LIN {X 0,Y 523.877,Z 238.227,A -85,B 0,C 180,E1 -4906.892,E2 -4906.892} C_VEL
LIN {X 0,Y 523.199,Z 238.314,A -85,B 0,C 180,E1 -4907.534,E2 -4907.534} C_VEL
LIN {X 0,Y 520.354,Z 238.667,A -85,B 0,C 180,E1 -4908.575,E2 -4908.575} C_VEL
LIN {X 0,Y 517.963,Z 238.966,A -85,B 0,C 180,E1 -4909.414,E2 -4909.414} C_VEL
LIN {X 0,Y 516.943,Z 239.092,A -85,B 0,C 180,E1 -4910.062,E2 -4910.062} C_VEL
LIN {X 0,Y 516.862,Z 239.1,A -85,B 0,C 180,E1 -4910.281,E2 -4910.281} C_VEL
LIN {X 0,Y 516.85,Z 239.107,A -85,B 0,C 180,E1 -4913.252,E2 -4913.252} C_VEL
LIN {X 0,Y 516.776,Z 239.117,A -85,B 0,C 180,E1 -4914.685,E2 -4914.685} C_VEL
LIN {X 0,Y 516.776,Z 242.58,A -85,B 0,C 180,E1 -4917.044,E2 -4917.044} C_VEL
LIN {X 0,Y 516.677,Z 246.727,A -85,B 0,C 180,E1 -4919.782,E2 -4919.782} C_VEL
LIN {X 0,Y 516.622,Z 250.843,A -85,B 0,C 180,E1 -4922.45,E2 -4922.45} C_VEL
LIN {X 0,Y 516.599,Z 255.972,A -85,B 0,C 180,E1 -4925.713,E2 -4925.713} C_VEL
LIN {X 0,Y 516.465,Z 260.373,A -85,B 0,C 180,E1 -4928.444,E2 -4928.444} C_VEL
LIN {X 0,Y 516.401,Z 264.484,A -85,B 0,C 180,E1 -4930.936,E2 -4930.936} C_VEL
LIN {X 0,Y 516.361,Z 268.626,A -85,B 0,C 180,E1 -4933.392,E2 -4933.392} C_VEL
LIN {X 0,Y 516.371,Z 273.427,A -85,B 0,C 180,E1 -4936.171,E2 -4936.171} C_VEL
LIN {X 0,Y 518.506,Z 285.677,A -85,B 0,C 180,E1 -4936.553,E2 -4936.553} C_VEL
LIN {X 0,Y 518.232,Z 298.164,A -85,B 0,C 180,E1 -4937.02,E2 -4937.02} C_VEL
LIN {X 0,Y 518.004,Z 310.503,A -85,B 0,C 180,E1 -4937.651,E2 -4937.651} C_VEL
LIN {X 0,Y 517.663,Z 322.372,A -85,B 0,C 180,E1 -4938.448,E2 -4938.448} C_VEL
LIN {X 0,Y 517.327,Z 332.848,A -85,B 0,C 180,E1 -4939.333,E2 -4939.333} C_VEL
LIN {X 0,Y 517.081,Z 341.406,A -85,B 0,C 180,E1 -4940.218,E2 -4940.218} C_VEL
LIN {X 0,Y 516.859,Z 349.287,A -85,B 0,C 180,E1 -4941.201,E2 -4941.201} C_VEL
LIN {X 0,Y 516.622,Z 356.995,A -85,B 0,C 180,E1 -4942.378,E2 -4942.378} C_VEL
LIN {X 0,Y 516.497,Z 364.061,A -85,B 0,C 180,E1 -4943.751,E2 -4943.751} C_VEL
LIN {X 0,Y 516.313,Z 368.775,A -85,B 0,C 180,E1 -4944.924,E2 -4944.924} C_VEL
LIN {X 0,Y 516.373,Z 372.379,A -85,B 0,C 180,E1 -4946.098,E2 -4946.098} C_VEL
LIN {X 0,Y 516.282,Z 374.246,A -85,B 0,C 180,E1 -4946.879,E2 -4946.879} C_VEL
LIN {X 0,Y 516.261,Z 375.654,A -85,B 0,C 180,E1 -4947.659,E2 -4947.659} C_VEL
LIN {X 0,Y 516.16,Z 377.273,A -85,B 0,C 180,E1 -4949.22,E2 -4949.22} C_VEL
LIN {X 0,Y 516.155,Z 377.51,A -85,B 0,C 180,E1 -4950,E2 -4950} C_VEL
LIN {X 0,Y 516.16,Z 377.327,A -85,B 0,C 180,E1 -4950.78,E2 -4950.78} C_VEL
LIN {X 0,Y 516.261,Z 375.779,A -85,B 0,C 180,E1 -4952.341,E2 -4952.341} C_VEL
LIN {X 0,Y 516.283,Z 374.426,A -85,B 0,C 180,E1 -4953.121,E2 -4953.121} C_VEL
LIN {X 0,Y 516.364,Z 371.563,A -85,B 0,C 180,E1 -4954.293,E2 -4954.293} C_VEL
LIN {X 0,Y 516.404,Z 367.684,A -85,B 0,C 180,E1 -4955.467,E2 -4955.467} C_VEL
LIN {X 0,Y 516.512,Z 362.677,A -85,B 0,C 180,E1 -4956.641,E2 -4956.641} C_VEL
LIN {X 0,Y 516.647,Z 356.375,A -85,B 0,C 180,E1 -4957.818,E2 -4957.818} C_VEL
LIN {X 0,Y 516.859,Z 348.484,A -85,B 0,C 180,E1 -4958.996,E2 -4958.996} C_VEL
LIN {X 0,Y 517.129,Z 338.665,A -85,B 0,C 180,E1 -4960.176,E2 -4960.176} C_VEL
LIN {X 0,Y 517.456,Z 328.368,A -85,B 0,C 180,E1 -4961.16,E2 -4961.16} C_VEL
LIN {X 0,Y 517.77,Z 317.683,A -85,B 0,C 180,E1 -4961.98,E2 -4961.98} C_VEL
LIN {X 0,Y 518.059,Z 307.006,A -85,B 0,C 180,E1 -4962.636,E2 -4962.636} C_VEL
LIN {X 0,Y 518.328,Z 294.474,A -85,B 0,C 180,E1 -4963.227,E2 -4963.227} C_VEL
LIN {X 0,Y 518.333,Z 284.206,A -85,B 0,C 180,E1 -4963.589,E2 -4963.589} C_VEL
LIN {X 0,Y 516.384,Z 273.353,A -85,B 0,C 180,E1 -4963.93,E2 -4963.93} C_VEL
LIN {X 0,Y 516.354,Z 268.778,A -85,B 0,C 180,E1 -4966.608,E2 -4966.608} C_VEL
LIN {X 0,Y 516.396,Z 264.635,A -85,B 0,C 180,E1 -4969.065,E2 -4969.065} C_VEL
LIN {X 0,Y 516.468,Z 260.521,A -85,B 0,C 180,E1 -4971.556,E2 -4971.556} C_VEL
LIN {X 0,Y 516.568,Z 256.141,A -85,B 0,C 180,E1 -4974.279,E2 -4974.279} C_VEL
LIN {X 0,Y 516.591,Z 252.355,A -85,B 0,C 180,E1 -4976.677,E2 -4976.677} C_VEL
LIN {X 0,Y 516.667,Z 248.011,A -85,B 0,C 180,E1 -4979.475,E2 -4979.475} C_VEL
LIN {X 0,Y 516.753,Z 243.385,A -85,B 0,C 180,E1 -4982.518,E2 -4982.518} C_VEL
LIN {X 0,Y 516.767,Z 239.227,A -85,B 0,C 180,E1 -4985.314,E2 -4985.314} C_VEL
LIN {X 0,Y 516.883,Z 239.097,A -85,B 0,C 180,E1 -4987.943,E2 -4987.943} C_VEL
LIN {X 0,Y 516.862,Z 239.103,A -85,B 0,C 180,E1 -4990.744,E2 -4990.744} C_VEL
LIN {X 0,Y 516.862,Z 239.105,A -85,B 0,C 180,E1 -4993.906,E2 -4993.906} C_VEL
LIN {X 0,Y 516.883,Z 239.1,A -85,B 0,C 180,E1 -4996.107,E2 -4996.107} C_VEL
LIN {X 0,Y 516.885,Z 239.101,A -85,B 0,C 180,E1 -4999.258,E2 -4999.258} C_VEL
LIN {X 0,Y 516.866,Z 239.105,A -85,B 0,C 180,E1 -5002.274,E2 -5002.274} C_VEL
LIN {X 0,Y 516.882,Z 239.097,A -85,B 0,C 180,E1 -5005.175,E2 -5005.175} C_VEL
LIN {X 0,Y 516.875,Z 239.101,A -85,B 0,C 180,E1 -5007.975,E2 -5007.975} C_VEL
LIN {X 0,Y 516.921,Z 239.097,A -85,B 0,C 180,E1 -5010.695,E2 -5010.695} C_VEL
LIN {X 0,Y 516.946,Z 239.092,A -85,B 0,C 180,E1 -5013.804,E2 -5013.804} C_VEL
LIN {X 0,Y 516.864,Z 239.1,A -85,B 0,C 180,E1 -5016.776,E2 -5016.776} C_VEL
LIN {X 0,Y 516.943,Z 239.093,A -85,B 0,C 180,E1 -5019.732,E2 -5019.732} C_VEL
LIN {X 0,Y 516.887,Z 239.1,A -85,B 0,C 180,E1 -5022.595,E2 -5022.595} C_VEL
LIN {X 0,Y 516.944,Z 239.093,A -85,B 0,C 180,E1 -5025.03,E2 -5025.03} C_VEL
LIN {X 0,Y 516.97,Z 239.091,A -85,B 0,C 180,E1 -5028.234,E2 -5028.234} C_VEL
LIN {X 0,Y 516.961,Z 239.094,A -85,B 0,C 180,E1 -5031.399,E2 -5031.399} C_VEL
LIN {X 0,Y 516.986,Z 239.085,A -85,B 0,C 180,E1 -5033.756,E2 -5033.756} C_VEL
LIN {X 0,Y 516.975,Z 239.09,A -85,B 0,C 180,E1 -5036.883,E2 -5036.883} C_VEL
LIN {X 0,Y 516.963,Z 239.093,A -85,B 0,C 180,E1 -5038.442,E2 -5038.442} C_VEL
LIN {X 0,Y 517.094,Z 239.073,A -85,B 0,C 180,E1 -5040.779,E2 -5040.779} C_VEL
LIN {X 0,Y 517.015,Z 239.085,A -85,B 0,C 180,E1 -5043.117,E2 -5043.117} C_VEL
LIN {X 0,Y 517.004,Z 239.083,A -85,B 0,C 180,E1 -5046.243,E2 -5046.243} C_VEL
LIN {X 0,Y 516.915,Z 239.092,A -85,B 0,C 180,E1 -5049.39,E2 -5049.39} C_VEL
LIN {X 0,Y 516.909,Z 239.096,A -85,B 0,C 180,E1 -5052.565,E2 -5052.565} C_VEL
LIN {X 0,Y 516.903,Z 239.099,A -85,B 0,C 180,E1 -5055.779,E2 -5055.779} C_VEL
LIN {X 0,Y 516.928,Z 239.093,A -85,B 0,C 180,E1 -5058.222,E2 -5058.222} C_VEL
LIN {X 0,Y 516.916,Z 239.097,A -85,B 0,C 180,E1 -5060.701,E2 -5060.701} C_VEL
LIN {X 0,Y 516.887,Z 239.103,A -85,B 0,C 180,E1 -5064.073,E2 -5064.073} C_VEL
LIN {X 0,Y 516.847,Z 239.102,A -85,B 0,C 180,E1 -5066.662,E2 -5066.662} C_VEL
LIN {X 0,Y 516.91,Z 239.098,A -85,B 0,C 180,E1 -5069.523,E2 -5069.523} C_VEL
LIN {X 0,Y 516.899,Z 239.1,A -85,B 0,C 180,E1 -5072.543,E2 -5072.543} C_VEL
LIN {X 0,Y 516.867,Z 239.101,A -85,B 0,C 180,E1 -5075.329,E2 -5075.329} C_VEL
LIN {X 0,Y 516.878,Z 239.101,A -85,B 0,C 180,E1 -5077.942,E2 -5077.942} C_VEL
LIN {X 0,Y 516.856,Z 239.102,A -85,B 0,C 180,E1 -5080.744,E2 -5080.744} C_VEL
LIN {X 0,Y 516.884,Z 239.099,A -85,B 0,C 180,E1 -5083.903,E2 -5083.903} C_VEL
LIN {X 0,Y 516.884,Z 239.103,A -85,B 0,C 180,E1 -5086.107,E2 -5086.107} C_VEL
LIN {X 0,Y 516.916,Z 239.098,A -85,B 0,C 180,E1 -5088.399,E2 -5088.399} C_VEL
LIN {X 0,Y 516.88,Z 239.103,A -85,B 0,C 180,E1 -5091.284,E2 -5091.284} C_VEL
LIN {X 0,Y 516.898,Z 239.131,A -85,B 0,C 180,E1 -5092.4,E2 -5092.4} C_VEL
LIN {X 0,Y 517.552,Z 243.857,A -85,B 0,C 180,E1 -5094.564,E2 -5094.564} C_VEL
LIN {X 0,Y 517.411,Z 250.474,A -85,B 0,C 180,E1 -5097.368,E2 -5097.368} C_VEL
LIN {X 0,Y 517.184,Z 258.699,A -85,B 0,C 180,E1 -5100.712,E2 -5100.712} C_VEL
LIN {X 0,Y 516.951,Z 267.651,A -85,B 0,C 180,E1 -5104.212,E2 -5104.212} C_VEL
LIN {X 0,Y 516.793,Z 275.509,A -85,B 0,C 180,E1 -5107.196,E2 -5107.196} C_VEL
LIN {X 0,Y 516.675,Z 283.353,A -85,B 0,C 180,E1 -5110.119,E2 -5110.119} C_VEL
LIN {X 0,Y 516.547,Z 291.134,A -85,B 0,C 180,E1 -5112.991,E2 -5112.991} C_VEL
LIN {X 0,Y 516.486,Z 299.991,A -85,B 0,C 180,E1 -5116.111,E2 -5116.111} C_VEL
LIN {X 0,Y 518.432,Z 313.144,A -85,B 0,C 180,E1 -5116.476,E2 -5116.476} C_VEL
LIN {X 0,Y 518.143,Z 326.477,A -85,B 0,C 180,E1 -5116.968,E2 -5116.968} C_VEL
LIN {X 0,Y 517.883,Z 337.839,A -85,B 0,C 180,E1 -5117.539,E2 -5117.539} C_VEL
LIN {X 0,Y 517.535,Z 348.884,A -85,B 0,C 180,E1 -5118.247,E2 -5118.247} C_VEL
LIN {X 0,Y 517.296,Z 359.799,A -85,B 0,C 180,E1 -5119.134,E2 -5119.134} C_VEL
LIN {X 0,Y 516.986,Z 368.698,A -85,B 0,C 180,E1 -5120.019,E2 -5120.019} C_VEL
LIN {X 0,Y 516.749,Z 378.37,A -85,B 0,C 180,E1 -5121.199,E2 -5121.199} C_VEL
LIN {X 0,Y 516.556,Z 386.069,A -85,B 0,C 180,E1 -5122.377,E2 -5122.377} C_VEL
LIN {X 0,Y 516.411,Z 393.166,A -85,B 0,C 180,E1 -5123.749,E2 -5123.749} C_VEL
LIN {X 0,Y 516.313,Z 397.887,A -85,B 0,C 180,E1 -5124.924,E2 -5124.924} C_VEL
LIN {X 0,Y 516.352,Z 401.496,A -85,B 0,C 180,E1 -5126.098,E2 -5126.098} C_VEL
LIN {X 0,Y 516.282,Z 403.355,A -85,B 0,C 180,E1 -5126.879,E2 -5126.879} C_VEL
LIN {X 0,Y 516.261,Z 404.75,A -85,B 0,C 180,E1 -5127.659,E2 -5127.659} C_VEL
LIN {X 0,Y 516.16,Z 406.351,A -85,B 0,C 180,E1 -5129.22,E2 -5129.22} C_VEL
LIN {X 0,Y 516.154,Z 406.567,A -85,B 0,C 180,E1 -5130,E2 -5130} C_VEL
LIN {X 0,Y 516.192,Z 405.746,A -85,B 0,C 180,E1 -5131.56,E2 -5131.56} C_VEL
LIN {X 0,Y 516.261,Z 404.753,A -85,B 0,C 180,E1 -5132.341,E2 -5132.341} C_VEL
LIN {X 0,Y 516.282,Z 403.359,A -85,B 0,C 180,E1 -5133.121,E2 -5133.121} C_VEL
LIN {X 0,Y 516.312,Z 400.426,A -85,B 0,C 180,E1 -5134.293,E2 -5134.293} C_VEL
LIN {X 0,Y 516.376,Z 396.455,A -85,B 0,C 180,E1 -5135.467,E2 -5135.467} C_VEL
LIN {X 0,Y 516.475,Z 390.583,A -85,B 0,C 180,E1 -5136.792,E2 -5136.792} C_VEL
LIN {X 0,Y 516.607,Z 383.671,A -85,B 0,C 180,E1 -5138.016,E2 -5138.016} C_VEL
LIN {X 0,Y 516.828,Z 375.389,A -85,B 0,C 180,E1 -5139.194,E2 -5139.194} C_VEL
LIN {X 0,Y 517.042,Z 366.9,A -85,B 0,C 180,E1 -5140.178,E2 -5140.178} C_VEL
LIN {X 0,Y 517.36,Z 356.412,A -85,B 0,C 180,E1 -5141.162,E2 -5141.162} C_VEL
LIN {X 0,Y 517.659,Z 345.376,A -85,B 0,C 180,E1 -5141.995,E2 -5141.995} C_VEL
LIN {X 0,Y 517.944,Z 334.663,A -85,B 0,C 180,E1 -5142.639,E2 -5142.639} C_VEL
LIN {X 0,Y 518.269,Z 323,A -85,B 0,C 180,E1 -5143.179,E2 -5143.179} C_VEL
LIN {X 0,Y 518.307,Z 311.386,A -85,B 0,C 180,E1 -5143.577,E2 -5143.577} C_VEL
LIN {X 0,Y 516.474,Z 299.802,A -85,B 0,C 180,E1 -5143.902,E2 -5143.902} C_VEL
LIN {X 0,Y 516.547,Z 291.136,A -85,B 0,C 180,E1 -5147.009,E2 -5147.009} C_VEL
LIN {X 0,Y 516.675,Z 283.353,A -85,B 0,C 180,E1 -5149.88,E2 -5149.88} C_VEL
LIN {X 0,Y 516.792,Z 275.509,A -85,B 0,C 180,E1 -5152.804,E2 -5152.804} C_VEL
LIN {X 0,Y 516.922,Z 268.768,A -85,B 0,C 180,E1 -5155.358,E2 -5155.358} C_VEL
LIN {X 0,Y 517.088,Z 260.928,A -85,B 0,C 180,E1 -5158.405,E2 -5158.405} C_VEL
LIN {X 0,Y 517.277,Z 254.107,A -85,B 0,C 180,E1 -5161.135,E2 -5161.135} C_VEL
LIN {X 0,Y 517.46,Z 247.579,A -85,B 0,C 180,E1 -5163.838,E2 -5163.838} C_VEL
LIN {X 0,Y 517.516,Z 243.189,A -85,B 0,C 180,E1 -5165.729,E2 -5165.729} C_VEL
LIN {X 0,Y 516.872,Z 239.104,A -85,B 0,C 180,E1 -5167.664,E2 -5167.664} C_VEL
LIN {X 0,Y 516.886,Z 239.103,A -85,B 0,C 180,E1 -5170.742,E2 -5170.742} C_VEL
LIN {X 0,Y 516.885,Z 239.099,A -85,B 0,C 180,E1 -5172.831,E2 -5172.831} C_VEL
LIN {X 0,Y 516.897,Z 239.099,A -85,B 0,C 180,E1 -5175.007,E2 -5175.007} C_VEL
LIN {X 0,Y 516.889,Z 239.098,A -85,B 0,C 180,E1 -5178.402,E2 -5178.402} C_VEL
LIN {X 0,Y 516.875,Z 239.098,A -85,B 0,C 180,E1 -5181.283,E2 -5181.283} C_VEL
LIN {X 0,Y 516.869,Z 239.104,A -85,B 0,C 180,E1 -5184.219,E2 -5184.219} C_VEL
LIN {X 0,Y 516.898,Z 239.099,A -85,B 0,C 180,E1 -5187.053,E2 -5187.053} C_VEL
LIN {X 0,Y 516.893,Z 239.098,A -85,B 0,C 180,E1 -5189.796,E2 -5189.796} C_VEL
LIN {X 0,Y 516.892,Z 239.103,A -85,B 0,C 180,E1 -5192.465,E2 -5192.465} C_VEL
LIN {X 0,Y 516.873,Z 239.1,A -85,B 0,C 180,E1 -5195.645,E2 -5195.645} C_VEL
LIN {X 0,Y 516.887,Z 239.097,A -85,B 0,C 180,E1 -5198.462,E2 -5198.462} C_VEL
LIN {X 0,Y 516.904,Z 239.099,A -85,B 0,C 180,E1 -5200.955,E2 -5200.955} C_VEL
LIN {X 0,Y 516.914,Z 239.096,A -85,B 0,C 180,E1 -5203.41,E2 -5203.41} C_VEL
LIN {X 0,Y 516.889,Z 239.099,A -85,B 0,C 180,E1 -5205.833,E2 -5205.833} C_VEL
LIN {X 0,Y 516.943,Z 239.09,A -85,B 0,C 180,E1 -5209.028,E2 -5209.028} C_VEL
LIN {X 0,Y 516.962,Z 239.088,A -85,B 0,C 180,E1 -5212.187,E2 -5212.187} C_VEL
LIN {X 0,Y 517.029,Z 239.082,A -85,B 0,C 180,E1 -5214.54,E2 -5214.54} C_VEL
LIN {X 0,Y 517.086,Z 239.074,A -85,B 0,C 180,E1 -5217.663,E2 -5217.663} C_VEL
LIN {X 0,Y 517.09,Z 239.073,A -85,B 0,C 180,E1 -5220.779,E2 -5220.779} C_VEL
LIN {X 0,Y 516.974,Z 239.09,A -85,B 0,C 180,E1 -5223.117,E2 -5223.117} C_VEL
LIN {X 0,Y 516.985,Z 239.085,A -85,B 0,C 180,E1 -5226.244,E2 -5226.244} C_VEL
LIN {X 0,Y 516.953,Z 239.089,A -85,B 0,C 180,E1 -5229.389,E2 -5229.389} C_VEL
LIN {X 0,Y 516.955,Z 239.093,A -85,B 0,C 180,E1 -5231.807,E2 -5231.807} C_VEL
LIN {X 0,Y 516.945,Z 239.094,A -85,B 0,C 180,E1 -5235.146,E2 -5235.146} C_VEL
LIN {X 0,Y 516.913,Z 239.095,A -85,B 0,C 180,E1 -5238.223,E2 -5238.223} C_VEL
LIN {X 0,Y 516.914,Z 239.098,A -85,B 0,C 180,E1 -5240.702,E2 -5240.702} C_VEL
LIN {X 0,Y 516.893,Z 239.102,A -85,B 0,C 180,E1 -5244.073,E2 -5244.073} C_VEL
LIN {X 0,Y 516.926,Z 239.093,A -85,B 0,C 180,E1 -5246.658,E2 -5246.658} C_VEL
LIN {X 0,Y 516.908,Z 239.098,A -85,B 0,C 180,E1 -5249.523,E2 -5249.523} C_VEL
LIN {X 0,Y 516.895,Z 239.101,A -85,B 0,C 180,E1 -5252.543,E2 -5252.543} C_VEL
LIN {X 0,Y 516.864,Z 239.1,A -85,B 0,C 180,E1 -5255.329,E2 -5255.329} C_VEL
LIN {X 0,Y 516.881,Z 239.102,A -85,B 0,C 180,E1 -5257.943,E2 -5257.943} C_VEL
LIN {X 0,Y 516.884,Z 239.1,A -85,B 0,C 180,E1 -5260.742,E2 -5260.742} C_VEL
LIN {X 0,Y 516.882,Z 239.099,A -85,B 0,C 180,E1 -5263.903,E2 -5263.903} C_VEL
LIN {X 0,Y 516.83,Z 239.104,A -85,B 0,C 180,E1 -5266.894,E2 -5266.894} C_VEL
LIN {X 0,Y 516.86,Z 239.106,A -85,B 0,C 180,E1 -5269.593,E2 -5269.593} C_VEL
LIN {X 0,Y 516.862,Z 239.1,A -85,B 0,C 180,E1 -5270.281,E2 -5270.281} C_VEL
LIN {X 0,Y 516.208,Z 239.183,A -85,B 0,C 180,E1 -5270.932,E2 -5270.932} C_VEL
LIN {X 0,Y 513.369,Z 239.537,A -85,B 0,C 180,E1 -5271.987,E2 -5271.987} C_VEL
LIN {X 0,Y 510.945,Z 239.841,A -85,B 0,C 180,E1 -5272.838,E2 -5272.838} C_VEL
LIN {X 0,Y 509.879,Z 239.974,A -85,B 0,C 180,E1 -5273.494,E2 -5273.494} C_VEL
LIN {X 0,Y 509.778,Z 239.985,A -85,B 0,C 180,E1 -5273.717,E2 -5273.717} C_VEL
LIN {X 0,Y 509.748,Z 239.992,A -85,B 0,C 180,E1 -5274.615,E2 -5274.615} C_VEL
LIN {X 0,Y 509.735,Z 244.044,A -85,B 0,C 180,E1 -5277.472,E2 -5277.472} C_VEL
LIN {X 0,Y 509.611,Z 248.339,A -85,B 0,C 180,E1 -5280.323,E2 -5280.323} C_VEL
LIN {X 0,Y 509.54,Z 252.321,A -85,B 0,C 180,E1 -5282.925,E2 -5282.925} C_VEL
LIN {X 0,Y 509.538,Z 256.418,A -85,B 0,C 180,E1 -5285.557,E2 -5285.557} C_VEL
LIN {X 0,Y 509.419,Z 260.501,A -85,B 0,C 180,E1 -5288.13,E2 -5288.13} C_VEL
LIN {X 0,Y 509.324,Z 264.603,A -85,B 0,C 180,E1 -5290.66,E2 -5290.66} C_VEL
LIN {X 0,Y 509.298,Z 268.769,A -85,B 0,C 180,E1 -5293.155,E2 -5293.155} C_VEL
LIN {X 0,Y 509.297,Z 273.583,A -85,B 0,C 180,E1 -5295.975,E2 -5295.975} C_VEL
LIN {X 0,Y 511.609,Z 286.656,A -85,B 0,C 180,E1 -5296.394,E2 -5296.394} C_VEL
LIN {X 0,Y 511.309,Z 299.505,A -85,B 0,C 180,E1 -5296.892,E2 -5296.892} C_VEL
LIN {X 0,Y 511.051,Z 311.483,A -85,B 0,C 180,E1 -5297.527,E2 -5297.527} C_VEL
LIN {X 0,Y 510.719,Z 322.58,A -85,B 0,C 180,E1 -5298.289,E2 -5298.289} C_VEL
LIN {X 0,Y 510.354,Z 333.055,A -85,B 0,C 180,E1 -5299.186,E2 -5299.186} C_VEL
LIN {X 0,Y 510.093,Z 341.611,A -85,B 0,C 180,E1 -5300.083,E2 -5300.083} C_VEL
LIN {X 0,Y 509.844,Z 349.492,A -85,B 0,C 180,E1 -5301.079,E2 -5301.079} C_VEL
LIN {X 0,Y 509.577,Z 357.199,A -85,B 0,C 180,E1 -5302.272,E2 -5302.272} C_VEL
LIN {X 0,Y 509.431,Z 364.264,A -85,B 0,C 180,E1 -5303.664,E2 -5303.664} C_VEL
LIN {X 0,Y 509.248,Z 368.976,A -85,B 0,C 180,E1 -5304.853,E2 -5304.853} C_VEL
LIN {X 0,Y 509.304,Z 372.58,A -85,B 0,C 180,E1 -5306.044,E2 -5306.044} C_VEL
LIN {X 0,Y 509.201,Z 374.447,A -85,B 0,C 180,E1 -5306.835,E2 -5306.835} C_VEL
LIN {X 0,Y 509.189,Z 375.854,A -85,B 0,C 180,E1 -5307.627,E2 -5307.627} C_VEL
LIN {X 0,Y 509.074,Z 377.473,A -85,B 0,C 180,E1 -5309.209,E2 -5309.209} C_VEL
LIN {X 0,Y 509.066,Z 377.71,A -85,B 0,C 180,E1 -5310,E2 -5310} C_VEL
LIN {X 0,Y 509.073,Z 377.526,A -85,B 0,C 180,E1 -5310.791,E2 -5310.791} C_VEL
LIN {X 0,Y 509.189,Z 375.977,A -85,B 0,C 180,E1 -5312.373,E2 -5312.373} C_VEL
LIN {X 0,Y 509.202,Z 374.624,A -85,B 0,C 180,E1 -5313.165,E2 -5313.165} C_VEL
LIN {X 0,Y 509.286,Z 371.762,A -85,B 0,C 180,E1 -5314.353,E2 -5314.353} C_VEL
LIN {X 0,Y 509.348,Z 367.881,A -85,B 0,C 180,E1 -5315.543,E2 -5315.543} C_VEL
LIN {X 0,Y 509.437,Z 362.159,A -85,B 0,C 180,E1 -5316.883,E2 -5316.883} C_VEL
LIN {X 0,Y 509.633,Z 355.349,A -85,B 0,C 180,E1 -5318.126,E2 -5318.126} C_VEL
LIN {X 0,Y 509.882,Z 347.201,A -85,B 0,C 180,E1 -5319.321,E2 -5319.321} C_VEL
LIN {X 0,Y 510.136,Z 338.86,A -85,B 0,C 180,E1 -5320.317,E2 -5320.317} C_VEL
LIN {X 0,Y 510.505,Z 328.56,A -85,B 0,C 180,E1 -5321.314,E2 -5321.314} C_VEL
LIN {X 0,Y 510.847,Z 317.412,A -85,B 0,C 180,E1 -5322.178,E2 -5322.178} C_VEL
LIN {X 0,Y 511.17,Z 305.38,A -85,B 0,C 180,E1 -5322.91,E2 -5322.91} C_VEL
LIN {X 0,Y 511.47,Z 293.358,A -85,B 0,C 180,E1 -5323.458,E2 -5323.458} C_VEL
LIN {X 0,Y 511.416,Z 284.798,A -85,B 0,C 180,E1 -5323.763,E2 -5323.763} C_VEL
LIN {X 0,Y 509.315,Z 273.557,A -85,B 0,C 180,E1 -5324.127,E2 -5324.127} C_VEL
LIN {X 0,Y 509.36,Z 267.527,A -85,B 0,C 180,E1 -5327.671,E2 -5327.671} C_VEL
LIN {X 0,Y 509.389,Z 262.007,A -85,B 0,C 180,E1 -5331.022,E2 -5331.022} C_VEL
LIN {X 0,Y 509.458,Z 257.927,A -85,B 0,C 180,E1 -5333.582,E2 -5333.582} C_VEL
LIN {X 0,Y 509.514,Z 253.692,A -85,B 0,C 180,E1 -5336.287,E2 -5336.287} C_VEL
LIN {X 0,Y 509.597,Z 249.719,A -85,B 0,C 180,E1 -5338.862,E2 -5338.862} C_VEL
LIN {X 0,Y 509.643,Z 245.581,A -85,B 0,C 180,E1 -5341.603,E2 -5341.603} C_VEL
LIN {X 0,Y 509.744,Z 241.398,A -85,B 0,C 180,E1 -5344.422,E2 -5344.422} C_VEL
LIN {X 0,Y 509.741,Z 240.007,A -85,B 0,C 180,E1 -5345.385,E2 -5345.385} C_VEL
LIN {X 0,Y 509.853,Z 239.976,A -85,B 0,C 180,E1 -5348.338,E2 -5348.338} C_VEL
LIN {X 0,Y 509.811,Z 239.979,A -85,B 0,C 180,E1 -5351.43,E2 -5351.43} C_VEL
LIN {X 0,Y 509.837,Z 239.976,A -85,B 0,C 180,E1 -5354.671,E2 -5354.671} C_VEL
LIN {X 0,Y 509.852,Z 239.975,A -85,B 0,C 180,E1 -5358.104,E2 -5358.104} C_VEL
LIN {X 0,Y 509.849,Z 239.979,A -85,B 0,C 180,E1 -5360.648,E2 -5360.648} C_VEL
LIN {X 0,Y 509.828,Z 239.978,A -85,B 0,C 180,E1 -5363.647,E2 -5363.647} C_VEL
LIN {X 0,Y 509.844,Z 239.975,A -85,B 0,C 180,E1 -5366.538,E2 -5366.538} C_VEL
LIN {X 0,Y 509.837,Z 239.98,A -85,B 0,C 180,E1 -5369.334,E2 -5369.334} C_VEL
LIN {X 0,Y 509.887,Z 239.971,A -85,B 0,C 180,E1 -5372.054,E2 -5372.054} C_VEL
LIN {X 0,Y 509.844,Z 239.977,A -85,B 0,C 180,E1 -5374.702,E2 -5374.702} C_VEL
LIN {X 0,Y 509.83,Z 239.979,A -85,B 0,C 180,E1 -5377.458,E2 -5377.458} C_VEL
LIN {X 0,Y 509.92,Z 239.967,A -85,B 0,C 180,E1 -5379.845,E2 -5379.845} C_VEL
LIN {X 0,Y 509.849,Z 239.978,A -85,B 0,C 180,E1 -5383.173,E2 -5383.173} C_VEL
LIN {X 0,Y 509.861,Z 239.974,A -85,B 0,C 180,E1 -5385.634,E2 -5385.634} C_VEL
LIN {X 0,Y 509.917,Z 239.967,A -85,B 0,C 180,E1 -5388.875,E2 -5388.875} C_VEL
LIN {X 0,Y 509.925,Z 239.965,A -85,B 0,C 180,E1 -5392.078,E2 -5392.078} C_VEL
LIN {X 0,Y 509.966,Z 239.96,A -85,B 0,C 180,E1 -5394.464,E2 -5394.464} C_VEL
LIN {X 0,Y 510.044,Z 239.95,A -85,B 0,C 180,E1 -5397.631,E2 -5397.631} C_VEL
LIN {X 0,Y 510.065,Z 239.948,A -85,B 0,C 180,E1 -5400.789,E2 -5400.789} C_VEL
LIN {X 0,Y 509.957,Z 239.964,A -85,B 0,C 180,E1 -5403.16,E2 -5403.16} C_VEL
LIN {X 0,Y 509.956,Z 239.962,A -85,B 0,C 180,E1 -5406.33,E2 -5406.33} C_VEL
LIN {X 0,Y 509.895,Z 239.972,A -85,B 0,C 180,E1 -5408.721,E2 -5408.721} C_VEL
LIN {X 0,Y 509.903,Z 239.971,A -85,B 0,C 180,E1 -5411.932,E2 -5411.932} C_VEL
LIN {X 0,Y 509.898,Z 239.971,A -85,B 0,C 180,E1 -5415.242,E2 -5415.242} C_VEL
LIN {X 0,Y 509.886,Z 239.971,A -85,B 0,C 180,E1 -5417.998,E2 -5417.998} C_VEL
LIN {X 0,Y 509.854,Z 239.976,A -85,B 0,C 180,E1 -5421.002,E2 -5421.002} C_VEL
LIN {X 0,Y 509.821,Z 239.978,A -85,B 0,C 180,E1 -5423.564,E2 -5423.564} C_VEL
LIN {X 0,Y 509.821,Z 239.978,A -85,B 0,C 180,E1 -5426.357,E2 -5426.357} C_VEL
LIN {X 0,Y 509.852,Z 239.976,A -85,B 0,C 180,E1 -5428.846,E2 -5428.846} C_VEL
LIN {X 0,Y 509.822,Z 239.979,A -85,B 0,C 180,E1 -5431.59,E2 -5431.59} C_VEL
LIN {X 0,Y 509.85,Z 239.977,A -85,B 0,C 180,E1 -5434.414,E2 -5434.414} C_VEL
LIN {X 0,Y 509.809,Z 239.981,A -85,B 0,C 180,E1 -5437.342,E2 -5437.342} C_VEL
LIN {X 0,Y 509.816,Z 239.977,A -85,B 0,C 180,E1 -5440.384,E2 -5440.384} C_VEL
LIN {X 0,Y 509.802,Z 239.985,A -85,B 0,C 180,E1 -5443.059,E2 -5443.059} C_VEL
LIN {X 0,Y 509.825,Z 239.979,A -85,B 0,C 180,E1 -5445.793,E2 -5445.793} C_VEL
LIN {X 0,Y 509.858,Z 239.976,A -85,B 0,C 180,E1 -5448.574,E2 -5448.574} C_VEL
LIN {X 0,Y 509.855,Z 239.979,A -85,B 0,C 180,E1 -5451.786,E2 -5451.786} C_VEL
LIN {X 0,Y 509.882,Z 240.168,A -85,B 0,C 180,E1 -5452.291,E2 -5452.291} C_VEL
LIN {X 0,Y 510.558,Z 245.333,A -85,B 0,C 180,E1 -5454.68,E2 -5454.68} C_VEL
LIN {X 0,Y 510.368,Z 251.947,A -85,B 0,C 180,E1 -5457.517,E2 -5457.517} C_VEL
LIN {X 0,Y 510.168,Z 259.721,A -85,B 0,C 180,E1 -5460.722,E2 -5460.722} C_VEL
LIN {X 0,Y 509.892,Z 268.662,A -85,B 0,C 180,E1 -5464.267,E2 -5464.267} C_VEL
LIN {X 0,Y 509.734,Z 276.513,A -85,B 0,C 180,E1 -5467.291,E2 -5467.291} C_VEL
LIN {X 0,Y 509.6,Z 284.359,A -85,B 0,C 180,E1 -5470.252,E2 -5470.252} C_VEL
LIN {X 0,Y 509.464,Z 293.248,A -85,B 0,C 180,E1 -5473.573,E2 -5473.573} C_VEL
LIN {X 0,Y 509.397,Z 299.786,A -85,B 0,C 180,E1 -5475.914,E2 -5475.914} C_VEL
LIN {X 0,Y 511.492,Z 312.943,A -85,B 0,C 180,E1 -5476.289,E2 -5476.289} C_VEL
LIN {X 0,Y 511.235,Z 326.277,A -85,B 0,C 180,E1 -5476.788,E2 -5476.788} C_VEL
LIN {X 0,Y 510.93,Z 337.664,A -85,B 0,C 180,E1 -5477.368,E2 -5477.368} C_VEL
LIN {X 0,Y 510.559,Z 348.684,A -85,B 0,C 180,E1 -5478.084,E2 -5478.084} C_VEL
LIN {X 0,Y 510.299,Z 359.599,A -85,B 0,C 180,E1 -5478.983,E2 -5478.983} C_VEL
LIN {X 0,Y 509.959,Z 368.498,A -85,B 0,C 180,E1 -5479.88,E2 -5479.88} C_VEL
LIN {X 0,Y 509.696,Z 378.169,A -85,B 0,C 180,E1 -5481.076,E2 -5481.076} C_VEL
LIN {X 0,Y 509.487,Z 385.868,A -85,B 0,C 180,E1 -5482.271,E2 -5482.271} C_VEL
LIN {X 0,Y 509.328,Z 392.058,A -85,B 0,C 180,E1 -5483.464,E2 -5483.464} C_VEL
LIN {X 0,Y 509.243,Z 397.687,A -85,B 0,C 180,E1 -5484.853,E2 -5484.853} C_VEL
LIN {X 0,Y 509.245,Z 401.296,A -85,B 0,C 180,E1 -5486.043,E2 -5486.043} C_VEL
LIN {X 0,Y 509.2,Z 403.156,A -85,B 0,C 180,E1 -5486.835,E2 -5486.835} C_VEL
LIN {X 0,Y 509.19,Z 404.551,A -85,B 0,C 180,E1 -5487.627,E2 -5487.627} C_VEL
LIN {X 0,Y 509.073,Z 406.151,A -85,B 0,C 180,E1 -5489.209,E2 -5489.209} C_VEL
LIN {X 0,Y 509.065,Z 406.368,A -85,B 0,C 180,E1 -5490,E2 -5490} C_VEL
LIN {X 0,Y 509.112,Z 405.547,A -85,B 0,C 180,E1 -5491.582,E2 -5491.582} C_VEL
LIN {X 0,Y 509.19,Z 404.554,A -85,B 0,C 180,E1 -5492.373,E2 -5492.373} C_VEL
LIN {X 0,Y 509.2,Z 403.16,A -85,B 0,C 180,E1 -5493.165,E2 -5493.165} C_VEL
LIN {X 0,Y 509.204,Z 400.225,A -85,B 0,C 180,E1 -5494.353,E2 -5494.353} C_VEL
LIN {X 0,Y 509.294,Z 396.254,A -85,B 0,C 180,E1 -5495.543,E2 -5495.543} C_VEL
LIN {X 0,Y 509.408,Z 390.248,A -85,B 0,C 180,E1 -5496.914,E2 -5496.914} C_VEL
LIN {X 0,Y 509.551,Z 383.471,A -85,B 0,C 180,E1 -5498.127,E2 -5498.127} C_VEL
LIN {X 0,Y 509.774,Z 375.188,A -85,B 0,C 180,E1 -5499.322,E2 -5499.322} C_VEL
LIN {X 0,Y 510.02,Z 366.7,A -85,B 0,C 180,E1 -5500.32,E2 -5500.32} C_VEL
LIN {X 0,Y 510.362,Z 356.212,A -85,B 0,C 180,E1 -5501.317,E2 -5501.317} C_VEL
LIN {X 0,Y 510.665,Z 345.175,A -85,B 0,C 180,E1 -5502.162,E2 -5502.162} C_VEL
LIN {X 0,Y 511,Z 334.462,A -85,B 0,C 180,E1 -5502.813,E2 -5502.813} C_VEL
LIN {X 0,Y 511.356,Z 322.8,A -85,B 0,C 180,E1 -5503.36,E2 -5503.36} C_VEL
LIN {X 0,Y 511.366,Z 312.1,A -85,B 0,C 180,E1 -5503.739,E2 -5503.739} C_VEL
LIN {X 0,Y 509.384,Z 299.596,A -85,B 0,C 180,E1 -5504.099,E2 -5504.099} C_VEL
LIN {X 0,Y 509.487,Z 290.994,A -85,B 0,C 180,E1 -5507.252,E2 -5507.252} C_VEL
LIN {X 0,Y 509.621,Z 282.841,A -85,B 0,C 180,E1 -5510.32,E2 -5510.32} C_VEL
LIN {X 0,Y 509.779,Z 275.388,A -85,B 0,C 180,E1 -5513.136,E2 -5513.136} C_VEL
LIN {X 0,Y 509.942,Z 266.987,A -85,B 0,C 180,E1 -5516.385,E2 -5516.385} C_VEL
LIN {X 0,Y 510.171,Z 258.461,A -85,B 0,C 180,E1 -5519.787,E2 -5519.787} C_VEL
LIN {X 0,Y 510.402,Z 251.018,A -85,B 0,C 180,E1 -5522.866,E2 -5522.866} C_VEL
LIN {X 0,Y 510.557,Z 245.322,A -85,B 0,C 180,E1 -5525.32,E2 -5525.32} C_VEL
LIN {X 0,Y 509.825,Z 239.982,A -85,B 0,C 180,E1 -5527.807,E2 -5527.807} C_VEL
LIN {X 0,Y 509.841,Z 239.981,A -85,B 0,C 180,E1 -5530.698,E2 -5530.698} C_VEL
LIN {X 0,Y 509.821,Z 239.984,A -85,B 0,C 180,E1 -5533.572,E2 -5533.572} C_VEL
LIN {X 0,Y 509.81,Z 239.98,A -85,B 0,C 180,E1 -5536.427,E2 -5536.427} C_VEL
LIN {X 0,Y 509.814,Z 239.979,A -85,B 0,C 180,E1 -5539.306,E2 -5539.306} C_VEL
LIN {X 0,Y 509.849,Z 239.974,A -85,B 0,C 180,E1 -5541.787,E2 -5541.787} C_VEL
LIN {X 0,Y 509.829,Z 239.978,A -85,B 0,C 180,E1 -5544.622,E2 -5544.622} C_VEL
LIN {X 0,Y 509.865,Z 239.976,A -85,B 0,C 180,E1 -5547.481,E2 -5547.481} C_VEL
LIN {X 0,Y 509.86,Z 239.974,A -85,B 0,C 180,E1 -5550.274,E2 -5550.274} C_VEL
LIN {X 0,Y 509.833,Z 239.978,A -85,B 0,C 180,E1 -5552.941,E2 -5552.941} C_VEL
LIN {X 0,Y 509.836,Z 239.976,A -85,B 0,C 180,E1 -5555.572,E2 -5555.572} C_VEL
LIN {X 0,Y 509.824,Z 239.979,A -85,B 0,C 180,E1 -5558.149,E2 -5558.149} C_VEL
LIN {X 0,Y 509.865,Z 239.974,A -85,B 0,C 180,E1 -5560.682,E2 -5560.682} C_VEL
LIN {X 0,Y 509.883,Z 239.974,A -85,B 0,C 180,E1 -5563.175,E2 -5563.175} C_VEL
LIN {X 0,Y 509.86,Z 239.974,A -85,B 0,C 180,E1 -5565.634,E2 -5565.634} C_VEL
LIN {X 0,Y 509.908,Z 239.966,A -85,B 0,C 180,E1 -5568.874,E2 -5568.874} C_VEL
LIN {X 0,Y 509.921,Z 239.965,A -85,B 0,C 180,E1 -5572.078,E2 -5572.078} C_VEL
LIN {X 0,Y 509.98,Z 239.96,A -85,B 0,C 180,E1 -5574.464,E2 -5574.464} C_VEL
LIN {X 0,Y 510.057,Z 239.95,A -85,B 0,C 180,E1 -5577.631,E2 -5577.631} C_VEL
LIN {X 0,Y 510.058,Z 239.952,A -85,B 0,C 180,E1 -5580,E2 -5580} C_VEL
LIN {X 0,Y 510.044,Z 239.95,A -85,B 0,C 180,E1 -5582.369,E2 -5582.369} C_VEL
LIN {X 0,Y 509.939,Z 239.963,A -85,B 0,C 180,E1 -5586.33,E2 -5586.33} C_VEL
LIN {X 0,Y 509.91,Z 239.972,A -85,B 0,C 180,E1 -5588.72,E2 -5588.72} C_VEL
LIN {X 0,Y 509.907,Z 239.97,A -85,B 0,C 180,E1 -5591.932,E2 -5591.932} C_VEL
LIN {X 0,Y 509.897,Z 239.973,A -85,B 0,C 180,E1 -5595.242,E2 -5595.242} C_VEL
LIN {X 0,Y 509.858,Z 239.975,A -85,B 0,C 180,E1 -5598.484,E2 -5598.484} C_VEL
LIN {X 0,Y 509.852,Z 239.974,A -85,B 0,C 180,E1 -5601.002,E2 -5601.002} C_VEL
LIN {X 0,Y 509.825,Z 239.979,A -85,B 0,C 180,E1 -5603.564,E2 -5603.564} C_VEL
LIN {X 0,Y 509.913,Z 239.967,A -85,B 0,C 180,E1 -5606.378,E2 -5606.378} C_VEL
LIN {X 0,Y 509.873,Z 239.975,A -85,B 0,C 180,E1 -5608.845,E2 -5608.845} C_VEL
LIN {X 0,Y 509.819,Z 239.978,A -85,B 0,C 180,E1 -5611.59,E2 -5611.59} C_VEL
LIN {X 0,Y 509.838,Z 239.979,A -85,B 0,C 180,E1 -5614.415,E2 -5614.415} C_VEL
LIN {X 0,Y 509.81,Z 239.98,A -85,B 0,C 180,E1 -5617.342,E2 -5617.342} C_VEL
LIN {X 0,Y 509.84,Z 239.976,A -85,B 0,C 180,E1 -5620.382,E2 -5620.382} C_VEL
LIN {X 0,Y 509.803,Z 239.984,A -85,B 0,C 180,E1 -5623.06,E2 -5623.06} C_VEL
LIN {X 0,Y 509.808,Z 239.982,A -85,B 0,C 180,E1 -5625.795,E2 -5625.795} C_VEL
LIN {X 0,Y 509.806,Z 239.98,A -85,B 0,C 180,E1 -5628.569,E2 -5628.569} C_VEL
LIN {X 0,Y 509.853,Z 239.975,A -85,B 0,C 180,E1 -5631.787,E2 -5631.787} C_VEL
LIN {X 0,Y 509.778,Z 239.985,A -85,B 0,C 180,E1 -5633.717,E2 -5633.717} C_VEL
LIN {X 0,Y 509.077,Z 240.26,A -85,B 0,C 180,E1 -5634.375,E2 -5634.375} C_VEL
LIN {X 0,Y 506.232,Z 241.577,A -85,B 0,C 180,E1 -5635.436,E2 -5635.436} C_VEL
LIN {X 0,Y 503.828,Z 243.04,A -85,B 0,C 180,E1 -5636.287,E2 -5636.287} C_VEL
LIN {X 0,Y 502.776,Z 244.124,A -85,B 0,C 180,E1 -5636.944,E2 -5636.944} C_VEL
LIN {X 0,Y 502.678,Z 244.457,A -85,B 0,C 180,E1 -5637.167,E2 -5637.167} C_VEL
LIN {X 0,Y 502.567,Z 248.813,A -85,B 0,C 180,E1 -5640.115,E2 -5640.115} C_VEL
LIN {X 0,Y 502.489,Z 252.435,A -85,B 0,C 180,E1 -5642.513,E2 -5642.513} C_VEL
LIN {X 0,Y 502.456,Z 256.852,A -85,B 0,C 180,E1 -5645.392,E2 -5645.392} C_VEL
LIN {X 0,Y 502.382,Z 260.634,A -85,B 0,C 180,E1 -5647.808,E2 -5647.808} C_VEL
LIN {X 0,Y 502.267,Z 264.742,A -85,B 0,C 180,E1 -5650.378,E2 -5650.378} C_VEL
LIN {X 0,Y 502.225,Z 268.901,A -85,B 0,C 180,E1 -5652.91,E2 -5652.91} C_VEL
LIN {X 0,Y 502.233,Z 273.729,A -85,B 0,C 180,E1 -5655.773,E2 -5655.773} C_VEL
LIN {X 0,Y 504.675,Z 286.876,A -85,B 0,C 180,E1 -5656.203,E2 -5656.203} C_VEL
LIN {X 0,Y 504.405,Z 299.719,A -85,B 0,C 180,E1 -5656.709,E2 -5656.709} C_VEL
LIN {X 0,Y 504.155,Z 311.31,A -85,B 0,C 180,E1 -5657.33,E2 -5657.33} C_VEL
LIN {X 0,Y 503.773,Z 322.788,A -85,B 0,C 180,E1 -5658.125,E2 -5658.125} C_VEL
LIN {X 0,Y 503.388,Z 333.261,A -85,B 0,C 180,E1 -5659.034,E2 -5659.034} C_VEL
LIN {X 0,Y 503.107,Z 341.817,A -85,B 0,C 180,E1 -5659.944,E2 -5659.944} C_VEL
LIN {X 0,Y 502.828,Z 349.696,A -85,B 0,C 180,E1 -5660.953,E2 -5660.953} C_VEL
LIN {X 0,Y 502.534,Z 357.402,A -85,B 0,C 180,E1 -5662.163,E2 -5662.163} C_VEL
LIN {X 0,Y 502.355,Z 364.468,A -85,B 0,C 180,E1 -5663.574,E2 -5663.574} C_VEL
LIN {X 0,Y 502.187,Z 369.178,A -85,B 0,C 180,E1 -5664.781,E2 -5664.781} C_VEL
LIN {X 0,Y 502.236,Z 372.781,A -85,B 0,C 180,E1 -5665.988,E2 -5665.988} C_VEL
LIN {X 0,Y 502.124,Z 374.648,A -85,B 0,C 180,E1 -5666.791,E2 -5666.791} C_VEL
LIN {X 0,Y 502.12,Z 376.054,A -85,B 0,C 180,E1 -5667.594,E2 -5667.594} C_VEL
LIN {X 0,Y 501.991,Z 377.672,A -85,B 0,C 180,E1 -5669.198,E2 -5669.198} C_VEL
LIN {X 0,Y 501.981,Z 377.909,A -85,B 0,C 180,E1 -5670,E2 -5670} C_VEL
LIN {X 0,Y 501.99,Z 377.725,A -85,B 0,C 180,E1 -5670.802,E2 -5670.802} C_VEL
LIN {X 0,Y 502.12,Z 376.176,A -85,B 0,C 180,E1 -5672.407,E2 -5672.407} C_VEL
LIN {X 0,Y 502.125,Z 374.822,A -85,B 0,C 180,E1 -5673.21,E2 -5673.21} C_VEL
LIN {X 0,Y 502.193,Z 371.96,A -85,B 0,C 180,E1 -5674.415,E2 -5674.415} C_VEL
LIN {X 0,Y 502.294,Z 368.078,A -85,B 0,C 180,E1 -5675.621,E2 -5675.621} C_VEL
LIN {X 0,Y 502.359,Z 363.073,A -85,B 0,C 180,E1 -5676.829,E2 -5676.829} C_VEL
LIN {X 0,Y 502.566,Z 356.768,A -85,B 0,C 180,E1 -5678.039,E2 -5678.039} C_VEL
LIN {X 0,Y 502.8,Z 348.875,A -85,B 0,C 180,E1 -5679.25,E2 -5679.25} C_VEL
LIN {X 0,Y 503.091,Z 340.828,A -85,B 0,C 180,E1 -5680.26,E2 -5680.26} C_VEL
LIN {X 0,Y 503.452,Z 331.006,A -85,B 0,C 180,E1 -5681.27,E2 -5681.27} C_VEL
LIN {X 0,Y 503.797,Z 321.345,A -85,B 0,C 180,E1 -5682.079,E2 -5682.079} C_VEL
LIN {X 0,Y 504.133,Z 310.403,A -85,B 0,C 180,E1 -5682.815,E2 -5682.815} C_VEL
LIN {X 0,Y 504.469,Z 298.32,A -85,B 0,C 180,E1 -5683.443,E2 -5683.443} C_VEL
LIN {X 0,Y 504.527,Z 285.747,A -85,B 0,C 180,E1 -5683.93,E2 -5683.93} C_VEL
LIN {X 0,Y 502.254,Z 273.705,A -85,B 0,C 180,E1 -5684.33,E2 -5684.33} C_VEL
LIN {X 0,Y 502.257,Z 267.666,A -85,B 0,C 180,E1 -5687.929,E2 -5687.929} C_VEL
LIN {X 0,Y 502.323,Z 263.504,A -85,B 0,C 180,E1 -5690.474,E2 -5690.474} C_VEL
LIN {X 0,Y 502.376,Z 259.419,A -85,B 0,C 180,E1 -5693.061,E2 -5693.061} C_VEL
LIN {X 0,Y 502.423,Z 255.32,A -85,B 0,C 180,E1 -5695.699,E2 -5695.699} C_VEL
LIN {X 0,Y 502.517,Z 251.201,A -85,B 0,C 180,E1 -5698.393,E2 -5698.393} C_VEL
LIN {X 0,Y 502.584,Z 246.621,A -85,B 0,C 180,E1 -5701.459,E2 -5701.459} C_VEL
LIN {X 0,Y 502.7,Z 242.275,A -85,B 0,C 180,E1 -5704.426,E2 -5704.426} C_VEL
LIN {X 0,Y 502.68,Z 241.485,A -85,B 0,C 180,E1 -5704.976,E2 -5704.976} C_VEL
LIN {X 0,Y 502.711,Z 240.864,A -85,B 0,C 180,E1 -5705.957,E2 -5705.957} C_VEL
LIN {X 0,Y 502.8,Z 240.854,A -85,B 0,C 180,E1 -5708.977,E2 -5708.977} C_VEL
LIN {X 0,Y 502.773,Z 240.861,A -85,B 0,C 180,E1 -5712.195,E2 -5712.195} C_VEL
LIN {X 0,Y 502.788,Z 240.857,A -85,B 0,C 180,E1 -5715.47,E2 -5715.47} C_VEL
LIN {X 0,Y 502.798,Z 240.854,A -85,B 0,C 180,E1 -5717.861,E2 -5717.861} C_VEL
LIN {X 0,Y 502.804,Z 240.853,A -85,B 0,C 180,E1 -5721.024,E2 -5721.024} C_VEL
LIN {X 0,Y 502.778,Z 240.86,A -85,B 0,C 180,E1 -5724.169,E2 -5724.169} C_VEL
LIN {X 0,Y 502.833,Z 240.849,A -85,B 0,C 180,E1 -5726.994,E2 -5726.994} C_VEL
LIN {X 0,Y 502.814,Z 240.851,A -85,B 0,C 180,E1 -5730.066,E2 -5730.066} C_VEL
LIN {X 0,Y 502.831,Z 240.852,A -85,B 0,C 180,E1 -5732.533,E2 -5732.533} C_VEL
LIN {X 0,Y 502.807,Z 240.852,A -85,B 0,C 180,E1 -5735.305,E2 -5735.305} C_VEL
LIN {X 0,Y 502.783,Z 240.859,A -85,B 0,C 180,E1 -5737.826,E2 -5737.826} C_VEL
LIN {X 0,Y 502.822,Z 240.849,A -85,B 0,C 180,E1 -5740.4,E2 -5740.4} C_VEL
LIN {X 0,Y 502.796,Z 240.857,A -85,B 0,C 180,E1 -5742.93,E2 -5742.93} C_VEL
LIN {X 0,Y 502.839,Z 240.849,A -85,B 0,C 180,E1 -5745.429,E2 -5745.429} C_VEL
LIN {X 0,Y 502.881,Z 240.844,A -85,B 0,C 180,E1 -5748.717,E2 -5748.717} C_VEL
LIN {X 0,Y 502.884,Z 240.843,A -85,B 0,C 180,E1 -5751.966,E2 -5751.966} C_VEL
LIN {X 0,Y 502.921,Z 240.837,A -85,B 0,C 180,E1 -5754.386,E2 -5754.386} C_VEL
LIN {X 0,Y 503.014,Z 240.826,A -85,B 0,C 180,E1 -5757.598,E2 -5757.598} C_VEL
LIN {X 0,Y 503.014,Z 240.827,A -85,B 0,C 180,E1 -5760.801,E2 -5760.801} C_VEL
LIN {X 0,Y 502.9,Z 240.844,A -85,B 0,C 180,E1 -5763.204,E2 -5763.204} C_VEL
LIN {X 0,Y 502.909,Z 240.84,A -85,B 0,C 180,E1 -5766.419,E2 -5766.419} C_VEL
LIN {X 0,Y 502.854,Z 240.848,A -85,B 0,C 180,E1 -5768.844,E2 -5768.844} C_VEL
LIN {X 0,Y 502.846,Z 240.852,A -85,B 0,C 180,E1 -5772.102,E2 -5772.102} C_VEL
LIN {X 0,Y 502.852,Z 240.849,A -85,B 0,C 180,E1 -5775.4,E2 -5775.4} C_VEL
LIN {X 0,Y 502.844,Z 240.848,A -85,B 0,C 180,E1 -5778.12,E2 -5778.12} C_VEL
LIN {X 0,Y 502.832,Z 240.853,A -85,B 0,C 180,E1 -5780.536,E2 -5780.536} C_VEL
LIN {X 0,Y 502.789,Z 240.853,A -85,B 0,C 180,E1 -5783.041,E2 -5783.041} C_VEL
LIN {X 0,Y 502.78,Z 240.859,A -85,B 0,C 180,E1 -5785.679,E2 -5785.679} C_VEL
LIN {X 0,Y 502.798,Z 240.853,A -85,B 0,C 180,E1 -5788.375,E2 -5788.375} C_VEL
LIN {X 0,Y 502.797,Z 240.857,A -85,B 0,C 180,E1 -5791.143,E2 -5791.143} C_VEL
LIN {X 0,Y 502.806,Z 240.855,A -85,B 0,C 180,E1 -5793.994,E2 -5793.994} C_VEL
LIN {X 0,Y 502.766,Z 240.857,A -85,B 0,C 180,E1 -5797.176,E2 -5797.176} C_VEL
LIN {X 0,Y 502.773,Z 240.855,A -85,B 0,C 180,E1 -5800.017,E2 -5800.017} C_VEL
LIN {X 0,Y 502.773,Z 240.856,A -85,B 0,C 180,E1 -5802.195,E2 -5802.195} C_VEL
LIN {X 0,Y 502.788,Z 240.855,A -85,B 0,C 180,E1 -5805.47,E2 -5805.47} C_VEL
LIN {X 0,Y 502.822,Z 240.852,A -85,B 0,C 180,E1 -5808.934,E2 -5808.934} C_VEL
LIN {X 0,Y 502.811,Z 240.935,A -85,B 0,C 180,E1 -5812.047,E2 -5812.047} C_VEL
LIN {X 0,Y 503.485,Z 245.277,A -85,B 0,C 180,E1 -5814.107,E2 -5814.107} C_VEL
LIN {X 0,Y 503.482,Z 249.669,A -85,B 0,C 180,E1 -5816.058,E2 -5816.058} C_VEL
LIN {X 0,Y 503.203,Z 256.296,A -85,B 0,C 180,E1 -5818.885,E2 -5818.885} C_VEL
LIN {X 0,Y 503.014,Z 263.043,A -85,B 0,C 180,E1 -5821.669,E2 -5821.669} C_VEL
LIN {X 0,Y 502.827,Z 270.785,A -85,B 0,C 180,E1 -5824.767,E2 -5824.767} C_VEL
LIN {X 0,Y 502.66,Z 278.63,A -85,B 0,C 180,E1 -5827.821,E2 -5827.821} C_VEL
LIN {X 0,Y 502.508,Z 286.45,A -85,B 0,C 180,E1 -5830.812,E2 -5830.812} C_VEL
LIN {X 0,Y 502.393,Z 294.219,A -85,B 0,C 180,E1 -5833.753,E2 -5833.753} C_VEL
LIN {X 0,Y 502.333,Z 299.581,A -85,B 0,C 180,E1 -5835.711,E2 -5835.711} C_VEL
LIN {X 0,Y 504.442,Z 312.739,A -85,B 0,C 180,E1 -5836.094,E2 -5836.094} C_VEL
LIN {X 0,Y 504.365,Z 324.947,A -85,B 0,C 180,E1 -5836.554,E2 -5836.554} C_VEL
LIN {X 0,Y 503.992,Z 336.03,A -85,B 0,C 180,E1 -5837.108,E2 -5837.108} C_VEL
LIN {X 0,Y 503.617,Z 347.286,A -85,B 0,C 180,E1 -5837.831,E2 -5837.831} C_VEL
LIN {X 0,Y 503.312,Z 358.325,A -85,B 0,C 180,E1 -5838.727,E2 -5838.727} C_VEL
LIN {X 0,Y 502.942,Z 368.297,A -85,B 0,C 180,E1 -5839.737,E2 -5839.737} C_VEL
LIN {X 0,Y 502.659,Z 377.969,A -85,B 0,C 180,E1 -5840.95,E2 -5840.95} C_VEL
LIN {X 0,Y 502.409,Z 385.667,A -85,B 0,C 180,E1 -5842.161,E2 -5842.161} C_VEL
LIN {X 0,Y 502.236,Z 392.356,A -85,B 0,C 180,E1 -5843.482,E2 -5843.482} C_VEL
LIN {X 0,Y 502.175,Z 397.487,A -85,B 0,C 180,E1 -5844.781,E2 -5844.781} C_VEL
LIN {X 0,Y 502.138,Z 401.095,A -85,B 0,C 180,E1 -5845.987,E2 -5845.987} C_VEL
LIN {X 0,Y 502.12,Z 402.956,A -85,B 0,C 180,E1 -5846.79,E2 -5846.79} C_VEL
LIN {X 0,Y 502.092,Z 404.351,A -85,B 0,C 180,E1 -5847.593,E2 -5847.593} C_VEL
LIN {X 0,Y 501.99,Z 405.952,A -85,B 0,C 180,E1 -5849.198,E2 -5849.198} C_VEL
LIN {X 0,Y 501.98,Z 406.168,A -85,B 0,C 180,E1 -5850,E2 -5850} C_VEL
LIN {X 0,Y 502.036,Z 405.347,A -85,B 0,C 180,E1 -5851.604,E2 -5851.604} C_VEL
LIN {X 0,Y 502.092,Z 404.354,A -85,B 0,C 180,E1 -5852.407,E2 -5852.407} C_VEL
LIN {X 0,Y 502.12,Z 402.96,A -85,B 0,C 180,E1 -5853.209,E2 -5853.209} C_VEL
LIN {X 0,Y 502.102,Z 400.025,A -85,B 0,C 180,E1 -5854.415,E2 -5854.415} C_VEL
LIN {X 0,Y 502.211,Z 396.054,A -85,B 0,C 180,E1 -5855.622,E2 -5855.622} C_VEL
LIN {X 0,Y 502.333,Z 390.047,A -85,B 0,C 180,E1 -5857.011,E2 -5857.011} C_VEL
LIN {X 0,Y 502.482,Z 383.27,A -85,B 0,C 180,E1 -5858.242,E2 -5858.242} C_VEL
LIN {X 0,Y 502.735,Z 374.987,A -85,B 0,C 180,E1 -5859.454,E2 -5859.454} C_VEL
LIN {X 0,Y 503,Z 366.499,A -85,B 0,C 180,E1 -5860.465,E2 -5860.465} C_VEL
LIN {X 0,Y 503.381,Z 356.011,A -85,B 0,C 180,E1 -5861.476,E2 -5861.476} C_VEL
LIN {X 0,Y 503.683,Z 344.974,A -85,B 0,C 180,E1 -5862.333,E2 -5862.333} C_VEL
LIN {X 0,Y 504.054,Z 334.262,A -85,B 0,C 180,E1 -5862.993,E2 -5862.993} C_VEL
LIN {X 0,Y 504.443,Z 322.6,A -85,B 0,C 180,E1 -5863.547,E2 -5863.547} C_VEL
LIN {X 0,Y 504.441,Z 312.735,A -85,B 0,C 180,E1 -5863.906,E2 -5863.906} C_VEL
LIN {X 0,Y 502.302,Z 299.39,A -85,B 0,C 180,E1 -5864.302,E2 -5864.302} C_VEL
LIN {X 0,Y 502.414,Z 291.997,A -85,B 0,C 180,E1 -5867.083,E2 -5867.083} C_VEL
LIN {X 0,Y 502.561,Z 284.243,A -85,B 0,C 180,E1 -5870.031,E2 -5870.031} C_VEL
LIN {X 0,Y 502.701,Z 276.379,A -85,B 0,C 180,E1 -5873.045,E2 -5873.045} C_VEL
LIN {X 0,Y 502.873,Z 268.539,A -85,B 0,C 180,E1 -5876.119,E2 -5876.119} C_VEL
LIN {X 0,Y 503.139,Z 260.73,A -85,B 0,C 180,E1 -5879.268,E2 -5879.268} C_VEL
LIN {X 0,Y 503.369,Z 252.965,A -85,B 0,C 180,E1 -5882.516,E2 -5882.516} C_VEL
LIN {X 0,Y 503.557,Z 246.36,A -85,B 0,C 180,E1 -5885.395,E2 -5885.395} C_VEL
LIN {X 0,Y 503.079,Z 242.431,A -85,B 0,C 180,E1 -5887.223,E2 -5887.223} C_VEL
LIN {X 0,Y 502.802,Z 240.857,A -85,B 0,C 180,E1 -5888.086,E2 -5888.086} C_VEL
LIN {X 0,Y 502.822,Z 240.854,A -85,B 0,C 180,E1 -5891.066,E2 -5891.066} C_VEL
LIN {X 0,Y 502.787,Z 240.855,A -85,B 0,C 180,E1 -5894.53,E2 -5894.53} C_VEL
LIN {X 0,Y 502.796,Z 240.853,A -85,B 0,C 180,E1 -5897.86,E2 -5897.86} C_VEL
LIN {X 0,Y 502.793,Z 240.854,A -85,B 0,C 180,E1 -5901.023,E2 -5901.023} C_VEL
LIN {X 0,Y 502.772,Z 240.861,A -85,B 0,C 180,E1 -5904.17,E2 -5904.17} C_VEL
LIN {X 0,Y 502.835,Z 240.851,A -85,B 0,C 180,E1 -5906.993,E2 -5906.993} C_VEL
LIN {X 0,Y 502.817,Z 240.851,A -85,B 0,C 180,E1 -5910.065,E2 -5910.065} C_VEL
LIN {X 0,Y 502.788,Z 240.858,A -85,B 0,C 180,E1 -5912.53,E2 -5912.53} C_VEL
LIN {X 0,Y 502.772,Z 240.855,A -85,B 0,C 180,E1 -5915.313,E2 -5915.313} C_VEL
LIN {X 0,Y 502.781,Z 240.86,A -85,B 0,C 180,E1 -5917.826,E2 -5917.826} C_VEL
LIN {X 0,Y 502.826,Z 240.85,A -85,B 0,C 180,E1 -5920.4,E2 -5920.4} C_VEL
LIN {X 0,Y 502.831,Z 240.852,A -85,B 0,C 180,E1 -5922.932,E2 -5922.932} C_VEL
LIN {X 0,Y 502.843,Z 240.848,A -85,B 0,C 180,E1 -5925.429,E2 -5925.429} C_VEL
LIN {X 0,Y 502.874,Z 240.843,A -85,B 0,C 180,E1 -5928.717,E2 -5928.717} C_VEL
LIN {X 0,Y 502.88,Z 240.843,A -85,B 0,C 180,E1 -5931.966,E2 -5931.966} C_VEL
LIN {X 0,Y 502.934,Z 240.837,A -85,B 0,C 180,E1 -5934.386,E2 -5934.386} C_VEL
LIN {X 0,Y 503.027,Z 240.825,A -85,B 0,C 180,E1 -5937.598,E2 -5937.598} C_VEL
LIN {X 0,Y 503.029,Z 240.827,A -85,B 0,C 180,E1 -5940,E2 -5940} C_VEL
LIN {X 0,Y 503.013,Z 240.826,A -85,B 0,C 180,E1 -5942.402,E2 -5942.402} C_VEL
LIN {X 0,Y 502.919,Z 240.837,A -85,B 0,C 180,E1 -5945.614,E2 -5945.614} C_VEL
LIN {X 0,Y 502.884,Z 240.843,A -85,B 0,C 180,E1 -5948.034,E2 -5948.034} C_VEL
LIN {X 0,Y 502.88,Z 240.843,A -85,B 0,C 180,E1 -5951.283,E2 -5951.283} C_VEL
LIN {X 0,Y 502.844,Z 240.848,A -85,B 0,C 180,E1 -5954.571,E2 -5954.571} C_VEL
LIN {X 0,Y 502.818,Z 240.85,A -85,B 0,C 180,E1 -5957.909,E2 -5957.909} C_VEL
LIN {X 0,Y 502.831,Z 240.854,A -85,B 0,C 180,E1 -5960.536,E2 -5960.536} C_VEL
LIN {X 0,Y 502.79,Z 240.853,A -85,B 0,C 180,E1 -5963.041,E2 -5963.041} C_VEL
LIN {X 0,Y 502.824,Z 240.853,A -85,B 0,C 180,E1 -5965.677,E2 -5965.677} C_VEL
LIN {X 0,Y 502.839,Z 240.849,A -85,B 0,C 180,E1 -5968.373,E2 -5968.373} C_VEL
LIN {X 0,Y 502.793,Z 240.854,A -85,B 0,C 180,E1 -5971.498,E2 -5971.498} C_VEL
LIN {X 0,Y 502.791,Z 240.856,A -85,B 0,C 180,E1 -5974.442,E2 -5974.442} C_VEL
LIN {X 0,Y 502.767,Z 240.857,A -85,B 0,C 180,E1 -5977.176,E2 -5977.176} C_VEL
LIN {X 0,Y 502.79,Z 240.855,A -85,B 0,C 180,E1 -5980.015,E2 -5980.015} C_VEL
LIN {X 0,Y 502.805,Z 240.853,A -85,B 0,C 180,E1 -5982.199,E2 -5982.199} C_VEL
LIN {X 0,Y 502.779,Z 240.856,A -85,B 0,C 180,E1 -5985.471,E2 -5985.471} C_VEL
LIN {X 0,Y 502.764,Z 240.856,A -85,B 0,C 180,E1 -5988.928,E2 -5988.928} C_VEL
LIN {X 0,Y 502.793,Z 240.853,A -85,B 0,C 180,E1 -5992.046,E2 -5992.046} C_VEL
LIN {X 0,Y 502.733,Z 240.862,A -85,B 0,C 180,E1 -5994.176,E2 -5994.176} C_VEL
LIN {X 0,Y 502.688,Z 241.346,A -85,B 0,C 180,E1 -5995.025,E2 -5995.025} C_VEL
LIN {X 0,Y 502.678,Z 244.457,A -85,B 0,C 180,E1 -5997.167,E2 -5997.167} C_VEL
LIN {X 0,Y 501.973,Z 245.496,A -85,B 0,C 180,E1 -5997.825,E2 -5997.825} C_VEL
LIN {X 0,Y 499.081,Z 247.393,A -85,B 0,C 180,E1 -5998.888,E2 -5998.888} C_VEL
LIN {X 0,Y 496.641,Z 248.933,A -85,B 0,C 180,E1 -5999.745,E2 -5999.745} C_VEL
LIN {X 0,Y 495.574,Z 250.034,A -85,B 0,C 180,E1 -6000.408,E2 -6000.408} C_VEL
LIN {X 0,Y 495.476,Z 250.378,A -85,B 0,C 180,E1 -6000.633,E2 -6000.633} C_VEL
LIN {X 0,Y 495.408,Z 254.44,A -85,B 0,C 180,E1 -6003.347,E2 -6003.347} C_VEL
LIN {X 0,Y 495.372,Z 258.034,A -85,B 0,C 180,E1 -6005.705,E2 -6005.705} C_VEL
LIN {X 0,Y 495.266,Z 262.137,A -85,B 0,C 180,E1 -6008.349,E2 -6008.349} C_VEL
LIN {X 0,Y 495.188,Z 266.279,A -85,B 0,C 180,E1 -6010.948,E2 -6010.948} C_VEL
LIN {X 0,Y 495.13,Z 270.446,A -85,B 0,C 180,E1 -6013.508,E2 -6013.508} C_VEL
LIN {X 0,Y 495.173,Z 273.898,A -85,B 0,C 180,E1 -6015.566,E2 -6015.566} C_VEL
LIN {X 0,Y 497.806,Z 287.854,A -85,B 0,C 180,E1 -6016.035,E2 -6016.035} C_VEL
LIN {X 0,Y 497.511,Z 299.933,A -85,B 0,C 180,E1 -6016.521,E2 -6016.521} C_VEL
LIN {X 0,Y 497.222,Z 311.526,A -85,B 0,C 180,E1 -6017.15,E2 -6017.15} C_VEL
LIN {X 0,Y 496.832,Z 322.996,A -85,B 0,C 180,E1 -6017.957,E2 -6017.957} C_VEL
LIN {X 0,Y 496.427,Z 333.467,A -85,B 0,C 180,E1 -6018.878,E2 -6018.878} C_VEL
LIN {X 0,Y 496.123,Z 342.022,A -85,B 0,C 180,E1 -6019.801,E2 -6019.801} C_VEL
LIN {X 0,Y 495.797,Z 349.902,A -85,B 0,C 180,E1 -6020.824,E2 -6020.824} C_VEL
LIN {X 0,Y 495.505,Z 357.606,A -85,B 0,C 180,E1 -6022.051,E2 -6022.051} C_VEL
LIN {X 0,Y 495.292,Z 364.67,A -85,B 0,C 180,E1 -6023.482,E2 -6023.482} C_VEL
LIN {X 0,Y 495.129,Z 369.38,A -85,B 0,C 180,E1 -6024.706,E2 -6024.706} C_VEL
LIN {X 0,Y 495.152,Z 372.983,A -85,B 0,C 180,E1 -6025.93,E2 -6025.93} C_VEL
LIN {X 0,Y 495.051,Z 374.849,A -85,B 0,C 180,E1 -6026.745,E2 -6026.745} C_VEL
LIN {X 0,Y 495.024,Z 376.254,A -85,B 0,C 180,E1 -6027.559,E2 -6027.559} C_VEL
LIN {X 0,Y 494.911,Z 377.872,A -85,B 0,C 180,E1 -6029.186,E2 -6029.186} C_VEL
LIN {X 0,Y 494.899,Z 378.109,A -85,B 0,C 180,E1 -6030,E2 -6030} C_VEL
LIN {X 0,Y 494.911,Z 377.924,A -85,B 0,C 180,E1 -6030.814,E2 -6030.814} C_VEL
LIN {X 0,Y 495.024,Z 376.375,A -85,B 0,C 180,E1 -6032.441,E2 -6032.441} C_VEL
LIN {X 0,Y 495.051,Z 375.021,A -85,B 0,C 180,E1 -6033.255,E2 -6033.255} C_VEL
LIN {X 0,Y 495.106,Z 372.158,A -85,B 0,C 180,E1 -6034.478,E2 -6034.478} C_VEL
LIN {X 0,Y 495.242,Z 368.275,A -85,B 0,C 180,E1 -6035.701,E2 -6035.701} C_VEL
LIN {X 0,Y 495.31,Z 363.27,A -85,B 0,C 180,E1 -6036.927,E2 -6036.927} C_VEL
LIN {X 0,Y 495.523,Z 356.964,A -85,B 0,C 180,E1 -6038.154,E2 -6038.154} C_VEL
LIN {X 0,Y 495.792,Z 349.07,A -85,B 0,C 180,E1 -6039.382,E2 -6039.382} C_VEL
LIN {X 0,Y 496.159,Z 339.248,A -85,B 0,C 180,E1 -6040.611,E2 -6040.611} C_VEL
LIN {X 0,Y 496.604,Z 328.944,A -85,B 0,C 180,E1 -6041.635,E2 -6041.635} C_VEL
LIN {X 0,Y 496.948,Z 318.332,A -85,B 0,C 180,E1 -6042.485,E2 -6042.485} C_VEL
LIN {X 0,Y 497.286,Z 307.572,A -85,B 0,C 180,E1 -6043.173,E2 -6043.173} C_VEL
LIN {X 0,Y 497.638,Z 295.023,A -85,B 0,C 180,E1 -6043.788,E2 -6043.788} C_VEL
LIN {X 0,Y 497.581,Z 286.31,A -85,B 0,C 180,E1 -6044.115,E2 -6044.115} C_VEL
LIN {X 0,Y 495.183,Z 273.872,A -85,B 0,C 180,E1 -6044.539,E2 -6044.539} C_VEL
LIN {X 0,Y 495.18,Z 267.82,A -85,B 0,C 180,E1 -6048.195,E2 -6048.195} C_VEL
LIN {X 0,Y 495.239,Z 263.646,A -85,B 0,C 180,E1 -6050.78,E2 -6050.78} C_VEL
LIN {X 0,Y 495.302,Z 259.557,A -85,B 0,C 180,E1 -6053.41,E2 -6053.41} C_VEL
LIN {X 0,Y 495.366,Z 255.451,A -85,B 0,C 180,E1 -6056.092,E2 -6056.092} C_VEL
LIN {X 0,Y 495.455,Z 251.31,A -85,B 0,C 180,E1 -6058.835,E2 -6058.835} C_VEL
LIN {X 0,Y 495.549,Z 247.097,A -85,B 0,C 180,E1 -6061.686,E2 -6061.686} C_VEL
LIN {X 0,Y 495.646,Z 242.794,A -85,B 0,C 180,E1 -6064.673,E2 -6064.673} C_VEL
LIN {X 0,Y 495.618,Z 241.751,A -85,B 0,C 180,E1 -6065.549,E2 -6065.549} C_VEL
LIN {X 0,Y 495.751,Z 241.735,A -85,B 0,C 180,E1 -6068.592,E2 -6068.592} C_VEL
LIN {X 0,Y 495.71,Z 241.735,A -85,B 0,C 180,E1 -6071.287,E2 -6071.287} C_VEL
LIN {X 0,Y 495.715,Z 241.74,A -85,B 0,C 180,E1 -6074.003,E2 -6074.003} C_VEL
LIN {X 0,Y 495.718,Z 241.738,A -85,B 0,C 180,E1 -6077.116,E2 -6077.116} C_VEL
LIN {X 0,Y 495.762,Z 241.73,A -85,B 0,C 180,E1 -6079.953,E2 -6079.953} C_VEL
LIN {X 0,Y 495.731,Z 241.735,A -85,B 0,C 180,E1 -6082.553,E2 -6082.553} C_VEL
LIN {X 0,Y 495.774,Z 241.728,A -85,B 0,C 180,E1 -6085.456,E2 -6085.456} C_VEL
LIN {X 0,Y 495.756,Z 241.73,A -85,B 0,C 180,E1 -6088.364,E2 -6088.364} C_VEL
LIN {X 0,Y 495.788,Z 241.728,A -85,B 0,C 180,E1 -6091.508,E2 -6091.508} C_VEL
LIN {X 0,Y 495.784,Z 241.729,A -85,B 0,C 180,E1 -6093.932,E2 -6093.932} C_VEL
LIN {X 0,Y 495.763,Z 241.729,A -85,B 0,C 180,E1 -6097.14,E2 -6097.14} C_VEL
LIN {X 0,Y 495.771,Z 241.727,A -85,B 0,C 180,E1 -6100.109,E2 -6100.109} C_VEL
LIN {X 0,Y 495.743,Z 241.733,A -85,B 0,C 180,E1 -6102.68,E2 -6102.68} C_VEL
LIN {X 0,Y 495.786,Z 241.728,A -85,B 0,C 180,E1 -6105.217,E2 -6105.217} C_VEL
LIN {X 0,Y 495.855,Z 241.72,A -85,B 0,C 180,E1 -6108.555,E2 -6108.555} C_VEL
LIN {X 0,Y 495.841,Z 241.72,A -85,B 0,C 180,E1 -6111.851,E2 -6111.851} C_VEL
LIN {X 0,Y 495.878,Z 241.714,A -85,B 0,C 180,E1 -6114.306,E2 -6114.306} C_VEL
LIN {X 0,Y 495.982,Z 241.702,A -85,B 0,C 180,E1 -6117.564,E2 -6117.564} C_VEL
LIN {X 0,Y 495.966,Z 241.705,A -85,B 0,C 180,E1 -6120.812,E2 -6120.812} C_VEL
LIN {X 0,Y 495.997,Z 241.701,A -85,B 0,C 180,E1 -6122.436,E2 -6122.436} C_VEL
LIN {X 0,Y 495.891,Z 241.714,A -85,B 0,C 180,E1 -6125.694,E2 -6125.694} C_VEL
LIN {X 0,Y 495.836,Z 241.721,A -85,B 0,C 180,E1 -6128.149,E2 -6128.149} C_VEL
LIN {X 0,Y 495.823,Z 241.722,A -85,B 0,C 180,E1 -6131.446,E2 -6131.446} C_VEL
LIN {X 0,Y 495.791,Z 241.727,A -85,B 0,C 180,E1 -6134.783,E2 -6134.783} C_VEL
LIN {X 0,Y 495.785,Z 241.729,A -85,B 0,C 180,E1 -6137.319,E2 -6137.319} C_VEL
LIN {X 0,Y 495.774,Z 241.729,A -85,B 0,C 180,E1 -6139.89,E2 -6139.89} C_VEL
LIN {X 0,Y 495.761,Z 241.729,A -85,B 0,C 180,E1 -6142.86,E2 -6142.86} C_VEL
LIN {X 0,Y 495.72,Z 241.736,A -85,B 0,C 180,E1 -6146.072,E2 -6146.072} C_VEL
LIN {X 0,Y 495.746,Z 241.733,A -85,B 0,C 180,E1 -6148.817,E2 -6148.817} C_VEL
LIN {X 0,Y 495.757,Z 241.731,A -85,B 0,C 180,E1 -6151.725,E2 -6151.725} C_VEL
LIN {X 0,Y 495.771,Z 241.73,A -85,B 0,C 180,E1 -6154.694,E2 -6154.694} C_VEL
LIN {X 0,Y 495.723,Z 241.738,A -85,B 0,C 180,E1 -6157.562,E2 -6157.562} C_VEL
LIN {X 0,Y 495.745,Z 241.731,A -85,B 0,C 180,E1 -6160.045,E2 -6160.045} C_VEL
LIN {X 0,Y 495.708,Z 241.74,A -85,B 0,C 180,E1 -6162.885,E2 -6162.885} C_VEL
LIN {X 0,Y 495.73,Z 241.737,A -85,B 0,C 180,E1 -6165.998,E2 -6165.998} C_VEL
LIN {X 0,Y 495.768,Z 241.732,A -85,B 0,C 180,E1 -6169.3,E2 -6169.3} C_VEL
LIN {X 0,Y 495.778,Z 241.831,A -85,B 0,C 180,E1 -6171.864,E2 -6171.864} C_VEL
LIN {X 0,Y 496.403,Z 245.849,A -85,B 0,C 180,E1 -6173.804,E2 -6173.804} C_VEL
LIN {X 0,Y 496.513,Z 249.598,A -85,B 0,C 180,E1 -6175.515,E2 -6175.515} C_VEL
LIN {X 0,Y 496.253,Z 256.215,A -85,B 0,C 180,E1 -6178.399,E2 -6178.399} C_VEL
LIN {X 0,Y 496.034,Z 262.863,A -85,B 0,C 180,E1 -6181.202,E2 -6181.202} C_VEL
LIN {X 0,Y 495.804,Z 270.672,A -85,B 0,C 180,E1 -6184.384,E2 -6184.384} C_VEL
LIN {X 0,Y 495.617,Z 278.5,A -85,B 0,C 180,E1 -6187.488,E2 -6187.488} C_VEL
LIN {X 0,Y 495.482,Z 285.2,A -85,B 0,C 180,E1 -6190.097,E2 -6190.097} C_VEL
LIN {X 0,Y 495.33,Z 292.956,A -85,B 0,C 180,E1 -6193.09,E2 -6193.09} C_VEL
LIN {X 0,Y 495.228,Z 299.375,A -85,B 0,C 180,E1 -6195.502,E2 -6195.502} C_VEL
LIN {X 0,Y 497.293,Z 312.531,A -85,B 0,C 180,E1 -6195.89,E2 -6195.89} C_VEL
LIN {X 0,Y 497.633,Z 316.361,A -85,B 0,C 180,E1 -6196.03,E2 -6196.03} C_VEL
LIN {X 0,Y 497.258,Z 329.153,A -85,B 0,C 180,E1 -6196.566,E2 -6196.566} C_VEL
LIN {X 0,Y 496.893,Z 340.787,A -85,B 0,C 180,E1 -6197.227,E2 -6197.227} C_VEL
LIN {X 0,Y 496.531,Z 350.893,A -85,B 0,C 180,E1 -6197.949,E2 -6197.949} C_VEL
LIN {X 0,Y 496.247,Z 361.344,A -85,B 0,C 180,E1 -6198.874,E2 -6198.874} C_VEL
LIN {X 0,Y 495.86,Z 369.884,A -85,B 0,C 180,E1 -6199.795,E2 -6199.795} C_VEL
LIN {X 0,Y 495.619,Z 377.768,A -85,B 0,C 180,E1 -6200.82,E2 -6200.82} C_VEL
LIN {X 0,Y 495.358,Z 385.467,A -85,B 0,C 180,E1 -6202.049,E2 -6202.049} C_VEL
LIN {X 0,Y 495.164,Z 392.564,A -85,B 0,C 180,E1 -6203.48,E2 -6203.48} C_VEL
LIN {X 0,Y 495.107,Z 397.287,A -85,B 0,C 180,E1 -6204.706,E2 -6204.706} C_VEL
LIN {X 0,Y 495.032,Z 400.894,A -85,B 0,C 180,E1 -6205.929,E2 -6205.929} C_VEL
LIN {X 0,Y 495.042,Z 402.756,A -85,B 0,C 180,E1 -6206.744,E2 -6206.744} C_VEL
LIN {X 0,Y 494.998,Z 404.151,A -85,B 0,C 180,E1 -6207.559,E2 -6207.559} C_VEL
LIN {X 0,Y 494.962,Z 405.146,A -85,B 0,C 180,E1 -6208.373,E2 -6208.373} C_VEL
LIN {X 0,Y 494.898,Z 405.969,A -85,B 0,C 180,E1 -6210,E2 -6210} C_VEL
LIN {X 0,Y 494.962,Z 405.148,A -85,B 0,C 180,E1 -6211.627,E2 -6211.627} C_VEL
LIN {X 0,Y 494.998,Z 404.154,A -85,B 0,C 180,E1 -6212.441,E2 -6212.441} C_VEL
LIN {X 0,Y 495.042,Z 402.76,A -85,B 0,C 180,E1 -6213.255,E2 -6213.255} C_VEL
LIN {X 0,Y 495.008,Z 399.824,A -85,B 0,C 180,E1 -6214.479,E2 -6214.479} C_VEL
LIN {X 0,Y 495.128,Z 395.854,A -85,B 0,C 180,E1 -6215.702,E2 -6215.702} C_VEL
LIN {X 0,Y 495.257,Z 389.745,A -85,B 0,C 180,E1 -6217.133,E2 -6217.133} C_VEL
LIN {X 0,Y 495.43,Z 383.069,A -85,B 0,C 180,E1 -6218.361,E2 -6218.361} C_VEL
LIN {X 0,Y 495.705,Z 374.787,A -85,B 0,C 180,E1 -6219.59,E2 -6219.59} C_VEL
LIN {X 0,Y 495.996,Z 366.298,A -85,B 0,C 180,E1 -6220.615,E2 -6220.615} C_VEL
LIN {X 0,Y 496.404,Z 355.811,A -85,B 0,C 180,E1 -6221.639,E2 -6221.639} C_VEL
LIN {X 0,Y 496.749,Z 344.581,A -85,B 0,C 180,E1 -6222.522,E2 -6222.522} C_VEL
LIN {X 0,Y 497.137,Z 334.062,A -85,B 0,C 180,E1 -6223.177,E2 -6223.177} C_VEL
LIN {X 0,Y 497.517,Z 322.4,A -85,B 0,C 180,E1 -6223.739,E2 -6223.739} C_VEL
LIN {X 0,Y 497.477,Z 313.68,A -85,B 0,C 180,E1 -6224.066,E2 -6224.066} C_VEL
LIN {X 0,Y 495.468,Z 300.863,A -85,B 0,C 180,E1 -6224.465,E2 -6224.465} C_VEL
LIN {X 0,Y 495.232,Z 299.194,A -85,B 0,C 180,E1 -6224.511,E2 -6224.511} C_VEL
LIN {X 0,Y 495.347,Z 291.847,A -85,B 0,C 180,E1 -6227.334,E2 -6227.334} C_VEL
LIN {X 0,Y 495.516,Z 283.423,A -85,B 0,C 180,E1 -6230.594,E2 -6230.594} C_VEL
LIN {X 0,Y 495.679,Z 276.253,A -85,B 0,C 180,E1 -6233.391,E2 -6233.391} C_VEL
LIN {X 0,Y 495.816,Z 269.539,A -85,B 0,C 180,E1 -6236.066,E2 -6236.066} C_VEL
LIN {X 0,Y 496.105,Z 261.744,A -85,B 0,C 180,E1 -6239.258,E2 -6239.258} C_VEL
LIN {X 0,Y 496.364,Z 253.983,A -85,B 0,C 180,E1 -6242.55,E2 -6242.55} C_VEL
LIN {X 0,Y 496.544,Z 247.389,A -85,B 0,C 180,E1 -6245.472,E2 -6245.472} C_VEL
LIN {X 0,Y 495.795,Z 241.951,A -85,B 0,C 180,E1 -6248.07,E2 -6248.07} C_VEL
LIN {X 0,Y 495.764,Z 241.733,A -85,B 0,C 180,E1 -6248.768,E2 -6248.768} C_VEL
LIN {X 0,Y 495.759,Z 241.735,A -85,B 0,C 180,E1 -6251.781,E2 -6251.781} C_VEL
LIN {X 0,Y 495.739,Z 241.736,A -85,B 0,C 180,E1 -6255.141,E2 -6255.141} C_VEL
LIN {X 0,Y 495.744,Z 241.732,A -85,B 0,C 180,E1 -6258.217,E2 -6258.217} C_VEL
LIN {X 0,Y 495.745,Z 241.73,A -85,B 0,C 180,E1 -6261.408,E2 -6261.408} C_VEL
LIN {X 0,Y 495.747,Z 241.733,A -85,B 0,C 180,E1 -6264.462,E2 -6264.462} C_VEL
LIN {X 0,Y 495.77,Z 241.731,A -85,B 0,C 180,E1 -6267.406,E2 -6267.406} C_VEL
LIN {X 0,Y 495.765,Z 241.73,A -85,B 0,C 180,E1 -6270.253,E2 -6270.253} C_VEL
LIN {X 0,Y 495.741,Z 241.732,A -85,B 0,C 180,E1 -6273.27,E2 -6273.27} C_VEL
LIN {X 0,Y 495.74,Z 241.731,A -85,B 0,C 180,E1 -6276.612,E2 -6276.612} C_VEL
LIN {X 0,Y 495.781,Z 241.729,A -85,B 0,C 180,E1 -6279.324,E2 -6279.324} C_VEL
LIN {X 0,Y 495.795,Z 241.726,A -85,B 0,C 180,E1 -6281.829,E2 -6281.829} C_VEL
LIN {X 0,Y 495.826,Z 241.724,A -85,B 0,C 180,E1 -6284.548,E2 -6284.548} C_VEL
LIN {X 0,Y 495.83,Z 241.725,A -85,B 0,C 180,E1 -6287.966,E2 -6287.966} C_VEL
LIN {X 0,Y 495.829,Z 241.721,A -85,B 0,C 180,E1 -6291.03,E2 -6291.03} C_VEL
LIN {X 0,Y 495.862,Z 241.719,A -85,B 0,C 180,E1 -6293.489,E2 -6293.489} C_VEL
LIN {X 0,Y 495.843,Z 241.723,A -85,B 0,C 180,E1 -6296.75,E2 -6296.75} C_VEL
LIN {X 0,Y 495.87,Z 241.718,A -85,B 0,C 180,E1 -6298.376,E2 -6298.376} C_VEL
LIN {X 0,Y 495.943,Z 241.707,A -85,B 0,C 180,E1 -6300.812,E2 -6300.812} C_VEL
LIN {X 0,Y 495.982,Z 241.702,A -85,B 0,C 180,E1 -6302.436,E2 -6302.436} C_VEL
LIN {X 0,Y 495.876,Z 241.714,A -85,B 0,C 180,E1 -6305.694,E2 -6305.694} C_VEL
LIN {X 0,Y 495.84,Z 241.72,A -85,B 0,C 180,E1 -6308.149,E2 -6308.149} C_VEL
LIN {X 0,Y 495.854,Z 241.719,A -85,B 0,C 180,E1 -6311.445,E2 -6311.445} C_VEL
LIN {X 0,Y 495.79,Z 241.727,A -85,B 0,C 180,E1 -6314.783,E2 -6314.783} C_VEL
LIN {X 0,Y 495.781,Z 241.727,A -85,B 0,C 180,E1 -6318.172,E2 -6318.172} C_VEL
LIN {X 0,Y 495.776,Z 241.73,A -85,B 0,C 180,E1 -6320.756,E2 -6320.756} C_VEL
LIN {X 0,Y 495.745,Z 241.732,A -85,B 0,C 180,E1 -6323.388,E2 -6323.388} C_VEL
LIN {X 0,Y 495.825,Z 241.723,A -85,B 0,C 180,E1 -6326.749,E2 -6326.749} C_VEL
LIN {X 0,Y 495.766,Z 241.73,A -85,B 0,C 180,E1 -6329.747,E2 -6329.747} C_VEL
LIN {X 0,Y 495.753,Z 241.733,A -85,B 0,C 180,E1 -6332.596,E2 -6332.596} C_VEL
LIN {X 0,Y 495.745,Z 241.731,A -85,B 0,C 180,E1 -6335.538,E2 -6335.538} C_VEL
LIN {X 0,Y 495.765,Z 241.729,A -85,B 0,C 180,E1 -6338.768,E2 -6338.768} C_VEL
LIN {X 0,Y 495.752,Z 241.732,A -85,B 0,C 180,E1 -6341.782,E2 -6341.782} C_VEL
LIN {X 0,Y 495.734,Z 241.734,A -85,B 0,C 180,E1 -6345.142,E2 -6345.142} C_VEL
LIN {X 0,Y 495.724,Z 241.736,A -85,B 0,C 180,E1 -6348.215,E2 -6348.215} C_VEL
LIN {X 0,Y 495.75,Z 241.736,A -85,B 0,C 180,E1 -6351.408,E2 -6351.408} C_VEL
LIN {X 0,Y 495.643,Z 241.747,A -85,B 0,C 180,E1 -6354.454,E2 -6354.454} C_VEL
LIN {X 0,Y 495.64,Z 244.231,A -85,B 0,C 180,E1 -6356.426,E2 -6356.426} C_VEL
LIN {X 0,Y 495.521,Z 248.405,A -85,B 0,C 180,E1 -6359.297,E2 -6359.297} C_VEL
LIN {X 0,Y 495.476,Z 250.378,A -85,B 0,C 180,E1 -6360.633,E2 -6360.633} C_VEL
LIN {X 0,Y 494.769,Z 251.448,A -85,B 0,C 180,E1 -6361.3,E2 -6361.3} C_VEL
LIN {X 0,Y 491.865,Z 253.366,A -85,B 0,C 180,E1 -6362.379,E2 -6362.379} C_VEL
LIN {X 0,Y 489.426,Z 254.92,A -85,B 0,C 180,E1 -6363.247,E2 -6363.247} C_VEL
LIN {X 0,Y 488.378,Z 256.038,A -85,B 0,C 180,E1 -6363.92,E2 -6363.92} C_VEL
LIN {X 0,Y 488.292,Z 256.391,A -85,B 0,C 180,E1 -6364.149,E2 -6364.149} C_VEL
LIN {X 0,Y 488.264,Z 259.542,A -85,B 0,C 180,E1 -6366.232,E2 -6366.232} C_VEL
LIN {X 0,Y 488.162,Z 264.361,A -85,B 0,C 180,E1 -6369.358,E2 -6369.358} C_VEL
LIN {X 0,Y 488.101,Z 269.22,A -85,B 0,C 180,E1 -6372.4,E2 -6372.4} C_VEL
LIN {X 0,Y 488.079,Z 274.083,A -85,B 0,C 180,E1 -6375.352,E2 -6375.352} C_VEL
LIN {X 0,Y 490.85,Z 288.452,A -85,B 0,C 180,E1 -6375.846,E2 -6375.846} C_VEL
LIN {X 0,Y 490.585,Z 301.255,A -85,B 0,C 180,E1 -6376.38,E2 -6376.38} C_VEL
LIN {X 0,Y 490.245,Z 313.189,A -85,B 0,C 180,E1 -6377.061,E2 -6377.061} C_VEL
LIN {X 0,Y 489.844,Z 324.489,A -85,B 0,C 180,E1 -6377.888,E2 -6377.888} C_VEL
LIN {X 0,Y 489.425,Z 334.735,A -85,B 0,C 180,E1 -6378.822,E2 -6378.822} C_VEL
LIN {X 0,Y 489.05,Z 343.926,A -85,B 0,C 180,E1 -6379.861,E2 -6379.861} C_VEL
LIN {X 0,Y 488.658,Z 352.847,A -85,B 0,C 180,E1 -6381.106,E2 -6381.106} C_VEL
LIN {X 0,Y 488.366,Z 360.029,A -85,B 0,C 180,E1 -6382.35,E2 -6382.35} C_VEL
LIN {X 0,Y 488.232,Z 365.816,A -85,B 0,C 180,E1 -6383.608,E2 -6383.608} C_VEL
LIN {X 0,Y 488.075,Z 369.582,A -85,B 0,C 180,E1 -6384.63,E2 -6384.63} C_VEL
LIN {X 0,Y 488.07,Z 373.184,A -85,B 0,C 180,E1 -6385.871,E2 -6385.871} C_VEL
LIN {X 0,Y 487.979,Z 375.049,A -85,B 0,C 180,E1 -6386.697,E2 -6386.697} C_VEL
LIN {X 0,Y 487.933,Z 376.455,A -85,B 0,C 180,E1 -6387.524,E2 -6387.524} C_VEL
LIN {X 0,Y 487.834,Z 378.072,A -85,B 0,C 180,E1 -6389.175,E2 -6389.175} C_VEL
LIN {X 0,Y 487.82,Z 378.308,A -85,B 0,C 180,E1 -6390,E2 -6390} C_VEL
LIN {X 0,Y 487.834,Z 378.123,A -85,B 0,C 180,E1 -6390.826,E2 -6390.826} C_VEL
LIN {X 0,Y 487.933,Z 376.573,A -85,B 0,C 180,E1 -6392.477,E2 -6392.477} C_VEL
LIN {X 0,Y 487.979,Z 375.219,A -85,B 0,C 180,E1 -6393.303,E2 -6393.303} C_VEL
LIN {X 0,Y 488.006,Z 372.357,A -85,B 0,C 180,E1 -6394.543,E2 -6394.543} C_VEL
LIN {X 0,Y 488.191,Z 368.472,A -85,B 0,C 180,E1 -6395.784,E2 -6395.784} C_VEL
LIN {X 0,Y 488.258,Z 363.467,A -85,B 0,C 180,E1 -6397.027,E2 -6397.027} C_VEL
LIN {X 0,Y 488.491,Z 357.16,A -85,B 0,C 180,E1 -6398.272,E2 -6398.272} C_VEL
LIN {X 0,Y 488.795,Z 349.265,A -85,B 0,C 180,E1 -6399.518,E2 -6399.518} C_VEL
LIN {X 0,Y 489.172,Z 339.443,A -85,B 0,C 180,E1 -6400.765,E2 -6400.765} C_VEL
LIN {X 0,Y 489.655,Z 329.137,A -85,B 0,C 180,E1 -6401.802,E2 -6401.802} C_VEL
LIN {X 0,Y 490.047,Z 317.488,A -85,B 0,C 180,E1 -6402.74,E2 -6402.74} C_VEL
LIN {X 0,Y 490.447,Z 305.943,A -85,B 0,C 180,E1 -6403.466,E2 -6403.466} C_VEL
LIN {X 0,Y 490.804,Z 293.91,A -85,B 0,C 180,E1 -6404.036,E2 -6404.036} C_VEL
LIN {X 0,Y 490.699,Z 287.254,A -85,B 0,C 180,E1 -6404.291,E2 -6404.291} C_VEL
LIN {X 0,Y 488.089,Z 274.056,A -85,B 0,C 180,E1 -6404.755,E2 -6404.755} C_VEL
LIN {X 0,Y 488.11,Z 268.5,A -85,B 0,C 180,E1 -6408.14,E2 -6408.14} C_VEL
LIN {X 0,Y 488.189,Z 263.792,A -85,B 0,C 180,E1 -6411.094,E2 -6411.094} C_VEL
LIN {X 0,Y 488.251,Z 259.687,A -85,B 0,C 180,E1 -6413.768,E2 -6413.768} C_VEL
LIN {X 0,Y 488.341,Z 255.058,A -85,B 0,C 180,E1 -6416.838,E2 -6416.838} C_VEL
LIN {X 0,Y 488.437,Z 251.421,A -85,B 0,C 180,E1 -6419.289,E2 -6419.289} C_VEL
LIN {X 0,Y 488.519,Z 247.256,A -85,B 0,C 180,E1 -6422.161,E2 -6422.161} C_VEL
LIN {X 0,Y 488.567,Z 243.052,A -85,B 0,C 180,E1 -6425.128,E2 -6425.128} C_VEL
LIN {X 0,Y 488.642,Z 242.618,A -85,B 0,C 180,E1 -6426.348,E2 -6426.348} C_VEL
LIN {X 0,Y 488.699,Z 242.608,A -85,B 0,C 180,E1 -6429.255,E2 -6429.255} C_VEL
LIN {X 0,Y 488.666,Z 242.615,A -85,B 0,C 180,E1 -6432.529,E2 -6432.529} C_VEL
LIN {X 0,Y 488.702,Z 242.611,A -85,B 0,C 180,E1 -6435.197,E2 -6435.197} C_VEL
LIN {X 0,Y 488.697,Z 242.613,A -85,B 0,C 180,E1 -6438.583,E2 -6438.583} C_VEL
LIN {X 0,Y 488.707,Z 242.609,A -85,B 0,C 180,E1 -6440.947,E2 -6440.947} C_VEL
LIN {X 0,Y 488.68,Z 242.614,A -85,B 0,C 180,E1 -6443.868,E2 -6443.868} C_VEL
LIN {X 0,Y 488.738,Z 242.604,A -85,B 0,C 180,E1 -6446.877,E2 -6446.877} C_VEL
LIN {X 0,Y 488.722,Z 242.608,A -85,B 0,C 180,E1 -6449.78,E2 -6449.78} C_VEL
LIN {X 0,Y 488.794,Z 242.6,A -85,B 0,C 180,E1 -6453.057,E2 -6453.057} C_VEL
LIN {X 0,Y 488.684,Z 242.613,A -85,B 0,C 180,E1 -6456.254,E2 -6456.254} C_VEL
LIN {X 0,Y 488.75,Z 242.604,A -85,B 0,C 180,E1 -6459.176,E2 -6459.176} C_VEL
LIN {X 0,Y 488.75,Z 242.604,A -85,B 0,C 180,E1 -6461.633,E2 -6461.633} C_VEL
LIN {X 0,Y 488.76,Z 242.605,A -85,B 0,C 180,E1 -6464.999,E2 -6464.999} C_VEL
LIN {X 0,Y 488.809,Z 242.598,A -85,B 0,C 180,E1 -6468.388,E2 -6468.388} C_VEL
LIN {X 0,Y 488.79,Z 242.599,A -85,B 0,C 180,E1 -6471.733,E2 -6471.733} C_VEL
LIN {X 0,Y 488.837,Z 242.59,A -85,B 0,C 180,E1 -6474.224,E2 -6474.224} C_VEL
LIN {X 0,Y 488.95,Z 242.578,A -85,B 0,C 180,E1 -6477.529,E2 -6477.529} C_VEL
LIN {X 0,Y 488.917,Z 242.583,A -85,B 0,C 180,E1 -6480.824,E2 -6480.824} C_VEL
LIN {X 0,Y 488.964,Z 242.577,A -85,B 0,C 180,E1 -6482.471,E2 -6482.471} C_VEL
LIN {X 0,Y 488.85,Z 242.591,A -85,B 0,C 180,E1 -6485.776,E2 -6485.776} C_VEL
LIN {X 0,Y 488.781,Z 242.601,A -85,B 0,C 180,E1 -6488.267,E2 -6488.267} C_VEL
LIN {X 0,Y 488.786,Z 242.599,A -85,B 0,C 180,E1 -6491.613,E2 -6491.613} C_VEL
LIN {X 0,Y 488.764,Z 242.603,A -85,B 0,C 180,E1 -6495,E2 -6495} C_VEL
LIN {X 0,Y 488.759,Z 242.604,A -85,B 0,C 180,E1 -6498.442,E2 -6498.442} C_VEL
LIN {X 0,Y 488.71,Z 242.609,A -85,B 0,C 180,E1 -6501.071,E2 -6501.071} C_VEL
LIN {X 0,Y 488.672,Z 242.614,A -85,B 0,C 180,E1 -6503.747,E2 -6503.747} C_VEL
LIN {X 0,Y 488.702,Z 242.609,A -85,B 0,C 180,E1 -6506.922,E2 -6506.922} C_VEL
LIN {X 0,Y 488.725,Z 242.607,A -85,B 0,C 180,E1 -6510.219,E2 -6510.219} C_VEL
LIN {X 0,Y 488.737,Z 242.605,A -85,B 0,C 180,E1 -6513.484,E2 -6513.484} C_VEL
LIN {X 0,Y 488.675,Z 242.613,A -85,B 0,C 180,E1 -6516.353,E2 -6516.353} C_VEL
LIN {X 0,Y 488.695,Z 242.613,A -85,B 0,C 180,E1 -6519.255,E2 -6519.255} C_VEL
LIN {X 0,Y 488.669,Z 242.614,A -85,B 0,C 180,E1 -6522.528,E2 -6522.528} C_VEL
LIN {X 0,Y 488.704,Z 242.61,A -85,B 0,C 180,E1 -6525.197,E2 -6525.197} C_VEL
LIN {X 0,Y 488.709,Z 242.612,A -85,B 0,C 180,E1 -6528.4,E2 -6528.4} C_VEL
LIN {X 0,Y 488.734,Z 242.61,A -85,B 0,C 180,E1 -6531.542,E2 -6531.542} C_VEL
LIN {X 0,Y 489.446,Z 247.35,A -85,B 0,C 180,E1 -6533.933,E2 -6533.933} C_VEL
LIN {X 0,Y 489.467,Z 251.731,A -85,B 0,C 180,E1 -6535.945,E2 -6535.945} C_VEL
LIN {X 0,Y 489.182,Z 258.331,A -85,B 0,C 180,E1 -6538.855,E2 -6538.855} C_VEL
LIN {X 0,Y 488.935,Z 264.979,A -85,B 0,C 180,E1 -6541.683,E2 -6541.683} C_VEL
LIN {X 0,Y 488.724,Z 272.913,A -85,B 0,C 180,E1 -6544.953,E2 -6544.953} C_VEL
LIN {X 0,Y 488.532,Z 280.602,A -85,B 0,C 180,E1 -6548.035,E2 -6548.035} C_VEL
LIN {X 0,Y 488.334,Z 288.37,A -85,B 0,C 180,E1 -6551.106,E2 -6551.106} C_VEL
LIN {X 0,Y 488.215,Z 296.078,A -85,B 0,C 180,E1 -6554.127,E2 -6554.127} C_VEL
LIN {X 0,Y 488.164,Z 299.177,A -85,B 0,C 180,E1 -6555.287,E2 -6555.287} C_VEL
LIN {X 0,Y 490.218,Z 312.328,A -85,B 0,C 180,E1 -6555.682,E2 -6555.682} C_VEL
LIN {X 0,Y 490.732,Z 316.926,A -85,B 0,C 180,E1 -6555.856,E2 -6555.856} C_VEL
LIN {X 0,Y 490.344,Z 328.954,A -85,B 0,C 180,E1 -6556.373,E2 -6556.373} C_VEL
LIN {X 0,Y 489.926,Z 341.15,A -85,B 0,C 180,E1 -6557.079,E2 -6557.079} C_VEL
LIN {X 0,Y 489.535,Z 351.988,A -85,B 0,C 180,E1 -6557.88,E2 -6557.88} C_VEL
LIN {X 0,Y 489.219,Z 362.189,A -85,B 0,C 180,E1 -6558.817,E2 -6558.817} C_VEL
LIN {X 0,Y 488.795,Z 371.364,A -85,B 0,C 180,E1 -6559.855,E2 -6559.855} C_VEL
LIN {X 0,Y 488.465,Z 380.307,A -85,B 0,C 180,E1 -6561.102,E2 -6561.102} C_VEL
LIN {X 0,Y 488.227,Z 387.505,A -85,B 0,C 180,E1 -6562.348,E2 -6562.348} C_VEL
LIN {X 0,Y 488.075,Z 392.849,A -85,B 0,C 180,E1 -6563.496,E2 -6563.496} C_VEL
LIN {X 0,Y 488.019,Z 397.087,A -85,B 0,C 180,E1 -6564.629,E2 -6564.629} C_VEL
LIN {X 0,Y 487.928,Z 400.694,A -85,B 0,C 180,E1 -6565.87,E2 -6565.87} C_VEL
LIN {X 0,Y 487.964,Z 402.557,A -85,B 0,C 180,E1 -6566.697,E2 -6566.697} C_VEL
LIN {X 0,Y 487.891,Z 404.947,A -85,B 0,C 180,E1 -6568.349,E2 -6568.349} C_VEL
LIN {X 0,Y 487.819,Z 405.77,A -85,B 0,C 180,E1 -6570,E2 -6570} C_VEL
LIN {X 0,Y 487.891,Z 404.949,A -85,B 0,C 180,E1 -6571.651,E2 -6571.651} C_VEL
LIN {X 0,Y 487.964,Z 402.561,A -85,B 0,C 180,E1 -6573.303,E2 -6573.303} C_VEL
LIN {X 0,Y 487.921,Z 399.624,A -85,B 0,C 180,E1 -6574.544,E2 -6574.544} C_VEL
LIN {X 0,Y 488.026,Z 395.653,A -85,B 0,C 180,E1 -6575.786,E2 -6575.786} C_VEL
LIN {X 0,Y 488.183,Z 389.545,A -85,B 0,C 180,E1 -6577.237,E2 -6577.237} C_VEL
LIN {X 0,Y 488.365,Z 382.868,A -85,B 0,C 180,E1 -6578.482,E2 -6578.482} C_VEL
LIN {X 0,Y 488.672,Z 374.586,A -85,B 0,C 180,E1 -6579.729,E2 -6579.729} C_VEL
LIN {X 0,Y 489.002,Z 366.098,A -85,B 0,C 180,E1 -6580.768,E2 -6580.768} C_VEL
LIN {X 0,Y 489.426,Z 355.61,A -85,B 0,C 180,E1 -6581.808,E2 -6581.808} C_VEL
LIN {X 0,Y 489.799,Z 344.36,A -85,B 0,C 180,E1 -6582.704,E2 -6582.704} C_VEL
LIN {X 0,Y 490.208,Z 333.861,A -85,B 0,C 180,E1 -6583.367,E2 -6583.367} C_VEL
LIN {X 0,Y 490.61,Z 322.198,A -85,B 0,C 180,E1 -6583.936,E2 -6583.936} C_VEL
LIN {X 0,Y 490.522,Z 314.239,A -85,B 0,C 180,E1 -6584.243,E2 -6584.243} C_VEL
LIN {X 0,Y 488.39,Z 300.725,A -85,B 0,C 180,E1 -6584.677,E2 -6584.677} C_VEL
LIN {X 0,Y 488.151,Z 299.008,A -85,B 0,C 180,E1 -6584.726,E2 -6584.726} C_VEL
LIN {X 0,Y 488.293,Z 291.687,A -85,B 0,C 180,E1 -6587.593,E2 -6587.593} C_VEL
LIN {X 0,Y 488.505,Z 282.839,A -85,B 0,C 180,E1 -6591.08,E2 -6591.08} C_VEL
LIN {X 0,Y 488.652,Z 274.997,A -85,B 0,C 180,E1 -6594.199,E2 -6594.199} C_VEL
LIN {X 0,Y 488.826,Z 268.245,A -85,B 0,C 180,E1 -6596.951,E2 -6596.951} C_VEL
LIN {X 0,Y 489.097,Z 261.642,A -85,B 0,C 180,E1 -6599.719,E2 -6599.719} C_VEL
LIN {X 0,Y 489.356,Z 254.997,A -85,B 0,C 180,E1 -6602.586,E2 -6602.586} C_VEL
LIN {X 0,Y 489.542,Z 249.436,A -85,B 0,C 180,E1 -6605.084,E2 -6605.084} C_VEL
LIN {X 0,Y 489.134,Z 245.143,A -85,B 0,C 180,E1 -6607.119,E2 -6607.119} C_VEL
LIN {X 0,Y 488.734,Z 242.61,A -85,B 0,C 180,E1 -6608.458,E2 -6608.458} C_VEL
LIN {X 0,Y 488.709,Z 242.613,A -85,B 0,C 180,E1 -6611.6,E2 -6611.6} C_VEL
LIN {X 0,Y 488.703,Z 242.61,A -85,B 0,C 180,E1 -6614.803,E2 -6614.803} C_VEL
LIN {X 0,Y 488.668,Z 242.614,A -85,B 0,C 180,E1 -6617.472,E2 -6617.472} C_VEL
LIN {X 0,Y 488.694,Z 242.613,A -85,B 0,C 180,E1 -6620.745,E2 -6620.745} C_VEL
LIN {X 0,Y 488.671,Z 242.615,A -85,B 0,C 180,E1 -6623.867,E2 -6623.867} C_VEL
LIN {X 0,Y 488.74,Z 242.606,A -85,B 0,C 180,E1 -6626.877,E2 -6626.877} C_VEL
LIN {X 0,Y 488.726,Z 242.607,A -85,B 0,C 180,E1 -6629.781,E2 -6629.781} C_VEL
LIN {X 0,Y 488.701,Z 242.609,A -85,B 0,C 180,E1 -6633.078,E2 -6633.078} C_VEL
LIN {X 0,Y 488.671,Z 242.615,A -85,B 0,C 180,E1 -6636.253,E2 -6636.253} C_VEL
LIN {X 0,Y 488.748,Z 242.604,A -85,B 0,C 180,E1 -6639.176,E2 -6639.176} C_VEL
LIN {X 0,Y 488.762,Z 242.604,A -85,B 0,C 180,E1 -6641.628,E2 -6641.628} C_VEL
LIN {X 0,Y 488.762,Z 242.604,A -85,B 0,C 180,E1 -6645,E2 -6645} C_VEL
LIN {X 0,Y 488.805,Z 242.596,A -85,B 0,C 180,E1 -6648.388,E2 -6648.388} C_VEL
LIN {X 0,Y 488.784,Z 242.601,A -85,B 0,C 180,E1 -6651.733,E2 -6651.733} C_VEL
LIN {X 0,Y 488.849,Z 242.591,A -85,B 0,C 180,E1 -6654.224,E2 -6654.224} C_VEL
LIN {X 0,Y 488.963,Z 242.577,A -85,B 0,C 180,E1 -6657.529,E2 -6657.529} C_VEL
LIN {X 0,Y 488.971,Z 242.578,A -85,B 0,C 180,E1 -6660,E2 -6660} C_VEL
LIN {X 0,Y 488.949,Z 242.578,A -85,B 0,C 180,E1 -6662.471,E2 -6662.471} C_VEL
LIN {X 0,Y 488.836,Z 242.591,A -85,B 0,C 180,E1 -6665.776,E2 -6665.776} C_VEL
LIN {X 0,Y 488.789,Z 242.599,A -85,B 0,C 180,E1 -6668.267,E2 -6668.267} C_VEL
LIN {X 0,Y 488.808,Z 242.598,A -85,B 0,C 180,E1 -6671.612,E2 -6671.612} C_VEL
LIN {X 0,Y 488.762,Z 242.604,A -85,B 0,C 180,E1 -6675,E2 -6675} C_VEL
LIN {X 0,Y 488.747,Z 242.605,A -85,B 0,C 180,E1 -6678.443,E2 -6678.443} C_VEL
LIN {X 0,Y 488.709,Z 242.607,A -85,B 0,C 180,E1 -6681.071,E2 -6681.071} C_VEL
LIN {X 0,Y 488.682,Z 242.613,A -85,B 0,C 180,E1 -6683.746,E2 -6683.746} C_VEL
LIN {X 0,Y 488.793,Z 242.6,A -85,B 0,C 180,E1 -6686.943,E2 -6686.943} C_VEL
LIN {X 0,Y 488.709,Z 242.61,A -85,B 0,C 180,E1 -6690.362,E2 -6690.362} C_VEL
LIN {X 0,Y 488.712,Z 242.607,A -85,B 0,C 180,E1 -6693.48,E2 -6693.48} C_VEL
LIN {X 0,Y 488.675,Z 242.613,A -85,B 0,C 180,E1 -6696.353,E2 -6696.353} C_VEL
LIN {X 0,Y 488.702,Z 242.611,A -85,B 0,C 180,E1 -6699.254,E2 -6699.254} C_VEL
LIN {X 0,Y 488.689,Z 242.613,A -85,B 0,C 180,E1 -6702.526,E2 -6702.526} C_VEL
LIN {X 0,Y 488.698,Z 242.61,A -85,B 0,C 180,E1 -6705.197,E2 -6705.197} C_VEL
LIN {X 0,Y 488.663,Z 242.614,A -85,B 0,C 180,E1 -6708.58,E2 -6708.58} C_VEL
LIN {X 0,Y 488.702,Z 242.608,A -85,B 0,C 180,E1 -6710.948,E2 -6710.948} C_VEL
LIN {X 0,Y 488.647,Z 242.617,A -85,B 0,C 180,E1 -6713.865,E2 -6713.865} C_VEL
LIN {X 0,Y 488.589,Z 243.204,A -85,B 0,C 180,E1 -6715.076,E2 -6715.076} C_VEL
LIN {X 0,Y 488.546,Z 247.46,A -85,B 0,C 180,E1 -6718.076,E2 -6718.076} C_VEL
LIN {X 0,Y 488.419,Z 252.25,A -85,B 0,C 180,E1 -6721.372,E2 -6721.372} C_VEL
LIN {X 0,Y 488.292,Z 256.391,A -85,B 0,C 180,E1 -6724.149,E2 -6724.149} C_VEL
LIN {X 0,Y 487.623,Z 257.481,A -85,B 0,C 180,E1 -6724.825,E2 -6724.825} C_VEL
LIN {X 0,Y 484.761,Z 259.417,A -85,B 0,C 180,E1 -6725.918,E2 -6725.918} C_VEL
LIN {X 0,Y 482.32,Z 260.983,A -85,B 0,C 180,E1 -6726.799,E2 -6726.799} C_VEL
LIN {X 0,Y 481.243,Z 262.115,A -85,B 0,C 180,E1 -6727.482,E2 -6727.482} C_VEL
LIN {X 0,Y 481.14,Z 262.476,A -85,B 0,C 180,E1 -6727.713,E2 -6727.713} C_VEL
LIN {X 0,Y 481.053,Z 266.593,A -85,B 0,C 180,E1 -6730.365,E2 -6730.365} C_VEL
LIN {X 0,Y 480.977,Z 270.785,A -85,B 0,C 180,E1 -6733.008,E2 -6733.008} C_VEL
LIN {X 0,Y 481.01,Z 274.266,A -85,B 0,C 180,E1 -6735.131,E2 -6735.131} C_VEL
LIN {X 0,Y 483.779,Z 288.292,A -85,B 0,C 180,E1 -6735.622,E2 -6735.622} C_VEL
LIN {X 0,Y 483.942,Z 294.494,A -85,B 0,C 180,E1 -6735.868,E2 -6735.868} C_VEL
LIN {X 0,Y 483.525,Z 306.435,A -85,B 0,C 180,E1 -6736.445,E2 -6736.445} C_VEL
LIN {X 0,Y 483.14,Z 318.741,A -85,B 0,C 180,E1 -6737.245,E2 -6737.245} C_VEL
LIN {X 0,Y 482.7,Z 329.509,A -85,B 0,C 180,E1 -6738.132,E2 -6738.132} C_VEL
LIN {X 0,Y 482.244,Z 338.845,A -85,B 0,C 180,E1 -6739.079,E2 -6739.079} C_VEL
LIN {X 0,Y 481.904,Z 347.351,A -85,B 0,C 180,E1 -6740.133,E2 -6740.133} C_VEL
LIN {X 0,Y 481.513,Z 355.613,A -85,B 0,C 180,E1 -6741.396,E2 -6741.396} C_VEL
LIN {X 0,Y 481.263,Z 362.267,A -85,B 0,C 180,E1 -6742.659,E2 -6742.659} C_VEL
LIN {X 0,Y 481.146,Z 368.362,A -85,B 0,C 180,E1 -6744.131,E2 -6744.131} C_VEL
LIN {X 0,Y 480.922,Z 372.325,A -85,B 0,C 180,E1 -6745.39,E2 -6745.39} C_VEL
LIN {X 0,Y 480.91,Z 375.25,A -85,B 0,C 180,E1 -6746.649,E2 -6746.649} C_VEL
LIN {X 0,Y 480.846,Z 376.656,A -85,B 0,C 180,E1 -6747.487,E2 -6747.487} C_VEL
LIN {X 0,Y 480.823,Z 377.654,A -85,B 0,C 180,E1 -6748.325,E2 -6748.325} C_VEL
LIN {X 0,Y 480.743,Z 378.507,A -85,B 0,C 180,E1 -6750,E2 -6750} C_VEL
LIN {X 0,Y 480.76,Z 378.322,A -85,B 0,C 180,E1 -6750.838,E2 -6750.838} C_VEL
LIN {X 0,Y 480.823,Z 377.737,A -85,B 0,C 180,E1 -6751.675,E2 -6751.675} C_VEL
LIN {X 0,Y 480.91,Z 375.417,A -85,B 0,C 180,E1 -6753.351,E2 -6753.351} C_VEL
LIN {X 0,Y 480.911,Z 372.556,A -85,B 0,C 180,E1 -6754.61,E2 -6754.61} C_VEL
LIN {X 0,Y 481.14,Z 368.67,A -85,B 0,C 180,E1 -6755.869,E2 -6755.869} C_VEL
LIN {X 0,Y 481.198,Z 363.663,A -85,B 0,C 180,E1 -6757.131,E2 -6757.131} C_VEL
LIN {X 0,Y 481.447,Z 357.358,A -85,B 0,C 180,E1 -6758.394,E2 -6758.394} C_VEL
LIN {X 0,Y 481.793,Z 349.461,A -85,B 0,C 180,E1 -6759.657,E2 -6759.657} C_VEL
LIN {X 0,Y 482.189,Z 339.639,A -85,B 0,C 180,E1 -6760.922,E2 -6760.922} C_VEL
LIN {X 0,Y 482.704,Z 329.331,A -85,B 0,C 180,E1 -6761.975,E2 -6761.975} C_VEL
LIN {X 0,Y 483.129,Z 317.616,A -85,B 0,C 180,E1 -6762.931,E2 -6762.931} C_VEL
LIN {X 0,Y 483.57,Z 306.133,A -85,B 0,C 180,E1 -6763.661,E2 -6763.661} C_VEL
LIN {X 0,Y 483.926,Z 294.098,A -85,B 0,C 180,E1 -6764.24,E2 -6764.24} C_VEL
LIN {X 0,Y 483.775,Z 288.202,A -85,B 0,C 180,E1 -6764.473,E2 -6764.473} C_VEL
LIN {X 0,Y 481.148,Z 275.089,A -85,B 0,C 180,E1 -6764.932,E2 -6764.932} C_VEL
LIN {X 0,Y 481.038,Z 274.236,A -85,B 0,C 180,E1 -6764.976,E2 -6764.976} C_VEL
LIN {X 0,Y 481.057,Z 268.141,A -85,B 0,C 180,E1 -6768.748,E2 -6768.748} C_VEL
LIN {X 0,Y 481.108,Z 263.941,A -85,B 0,C 180,E1 -6771.42,E2 -6771.42} C_VEL
LIN {X 0,Y 481.203,Z 259.827,A -85,B 0,C 180,E1 -6774.139,E2 -6774.139} C_VEL
LIN {X 0,Y 481.281,Z 255.526,A -85,B 0,C 180,E1 -6777.03,E2 -6777.03} C_VEL
LIN {X 0,Y 481.402,Z 251.531,A -85,B 0,C 180,E1 -6779.76,E2 -6779.76} C_VEL
LIN {X 0,Y 481.485,Z 247.343,A -85,B 0,C 180,E1 -6782.689,E2 -6782.689} C_VEL
LIN {X 0,Y 481.517,Z 243.875,A -85,B 0,C 180,E1 -6785.179,E2 -6785.179} C_VEL
LIN {X 0,Y 481.523,Z 243.505,A -85,B 0,C 180,E1 -6785.72,E2 -6785.72} C_VEL
LIN {X 0,Y 481.671,Z 243.487,A -85,B 0,C 180,E1 -6788.859,E2 -6788.859} C_VEL
LIN {X 0,Y 481.625,Z 243.494,A -85,B 0,C 180,E1 -6792.163,E2 -6792.163} C_VEL
LIN {X 0,Y 481.656,Z 243.489,A -85,B 0,C 180,E1 -6795.542,E2 -6795.542} C_VEL
LIN {X 0,Y 481.652,Z 243.489,A -85,B 0,C 180,E1 -6798.957,E2 -6798.957} C_VEL
LIN {X 0,Y 481.658,Z 243.488,A -85,B 0,C 180,E1 -6801.993,E2 -6801.993} C_VEL
LIN {X 0,Y 481.687,Z 243.482,A -85,B 0,C 180,E1 -6805.318,E2 -6805.318} C_VEL
LIN {X 0,Y 481.646,Z 243.488,A -85,B 0,C 180,E1 -6808.311,E2 -6808.311} C_VEL
LIN {X 0,Y 481.7,Z 243.484,A -85,B 0,C 180,E1 -6811.218,E2 -6811.218} C_VEL
LIN {X 0,Y 481.693,Z 243.486,A -85,B 0,C 180,E1 -6814.042,E2 -6814.042} C_VEL
LIN {X 0,Y 481.677,Z 243.484,A -85,B 0,C 180,E1 -6816.812,E2 -6816.812} C_VEL
LIN {X 0,Y 481.698,Z 243.486,A -85,B 0,C 180,E1 -6819.503,E2 -6819.503} C_VEL
LIN {X 0,Y 481.684,Z 243.483,A -85,B 0,C 180,E1 -6822.157,E2 -6822.157} C_VEL
LIN {X 0,Y 481.743,Z 243.479,A -85,B 0,C 180,E1 -6824.776,E2 -6824.776} C_VEL
LIN {X 0,Y 481.755,Z 243.476,A -85,B 0,C 180,E1 -6828.215,E2 -6828.215} C_VEL
LIN {X 0,Y 481.744,Z 243.478,A -85,B 0,C 180,E1 -6831.611,E2 -6831.611} C_VEL
LIN {X 0,Y 481.799,Z 243.467,A -85,B 0,C 180,E1 -6834.139,E2 -6834.139} C_VEL
LIN {X 0,Y 481.916,Z 243.454,A -85,B 0,C 180,E1 -6837.492,E2 -6837.492} C_VEL
LIN {X 0,Y 481.87,Z 243.461,A -85,B 0,C 180,E1 -6840.836,E2 -6840.836} C_VEL
LIN {X 0,Y 481.931,Z 243.454,A -85,B 0,C 180,E1 -6842.507,E2 -6842.507} C_VEL
LIN {X 0,Y 481.81,Z 243.468,A -85,B 0,C 180,E1 -6845.86,E2 -6845.86} C_VEL
LIN {X 0,Y 481.734,Z 243.48,A -85,B 0,C 180,E1 -6848.389,E2 -6848.389} C_VEL
LIN {X 0,Y 481.737,Z 243.477,A -85,B 0,C 180,E1 -6851.785,E2 -6851.785} C_VEL
LIN {X 0,Y 481.745,Z 243.477,A -85,B 0,C 180,E1 -6855.224,E2 -6855.224} C_VEL
LIN {X 0,Y 481.716,Z 243.482,A -85,B 0,C 180,E1 -6858.722,E2 -6858.722} C_VEL
LIN {X 0,Y 481.649,Z 243.488,A -85,B 0,C 180,E1 -6861.395,E2 -6861.395} C_VEL
LIN {X 0,Y 481.651,Z 243.491,A -85,B 0,C 180,E1 -6864.115,E2 -6864.115} C_VEL
LIN {X 0,Y 481.677,Z 243.485,A -85,B 0,C 180,E1 -6867.122,E2 -6867.122} C_VEL
LIN {X 0,Y 481.674,Z 243.486,A -85,B 0,C 180,E1 -6869.741,E2 -6869.741} C_VEL
LIN {X 0,Y 481.675,Z 243.486,A -85,B 0,C 180,E1 -6872.674,E2 -6872.674} C_VEL
LIN {X 0,Y 481.663,Z 243.486,A -85,B 0,C 180,E1 -6875.204,E2 -6875.204} C_VEL
LIN {X 0,Y 481.667,Z 243.485,A -85,B 0,C 180,E1 -6878.86,E2 -6878.86} C_VEL
LIN {X 0,Y 481.631,Z 243.49,A -85,B 0,C 180,E1 -6882.163,E2 -6882.163} C_VEL
LIN {X 0,Y 481.657,Z 243.488,A -85,B 0,C 180,E1 -6885.542,E2 -6885.542} C_VEL
LIN {X 0,Y 481.659,Z 243.489,A -85,B 0,C 180,E1 -6888.958,E2 -6888.958} C_VEL
LIN {X 0,Y 481.719,Z 243.614,A -85,B 0,C 180,E1 -6891.48,E2 -6891.48} C_VEL
LIN {X 0,Y 482.425,Z 248.373,A -85,B 0,C 180,E1 -6893.842,E2 -6893.842} C_VEL
LIN {X 0,Y 482.448,Z 253.282,A -85,B 0,C 180,E1 -6896.134,E2 -6896.134} C_VEL
LIN {X 0,Y 482.176,Z 259.343,A -85,B 0,C 180,E1 -6898.84,E2 -6898.84} C_VEL
LIN {X 0,Y 481.894,Z 265.978,A -85,B 0,C 180,E1 -6901.707,E2 -6901.707} C_VEL
LIN {X 0,Y 481.676,Z 273.768,A -85,B 0,C 180,E1 -6904.967,E2 -6904.967} C_VEL
LIN {X 0,Y 481.471,Z 281.577,A -85,B 0,C 180,E1 -6908.147,E2 -6908.147} C_VEL
LIN {X 0,Y 481.252,Z 289.315,A -85,B 0,C 180,E1 -6911.26,E2 -6911.26} C_VEL
LIN {X 0,Y 481.144,Z 295.904,A -85,B 0,C 180,E1 -6913.887,E2 -6913.887} C_VEL
LIN {X 0,Y 481.097,Z 298.982,A -85,B 0,C 180,E1 -6915.066,E2 -6915.066} C_VEL
LIN {X 0,Y 483.156,Z 312.128,A -85,B 0,C 180,E1 -6915.468,E2 -6915.468} C_VEL
LIN {X 0,Y 483.832,Z 316.73,A -85,B 0,C 180,E1 -6915.65,E2 -6915.65} C_VEL
LIN {X 0,Y 483.448,Z 328.757,A -85,B 0,C 180,E1 -6916.175,E2 -6916.175} C_VEL
LIN {X 0,Y 483.008,Z 340.952,A -85,B 0,C 180,E1 -6916.891,E2 -6916.891} C_VEL
LIN {X 0,Y 482.531,Z 351.414,A -85,B 0,C 180,E1 -6917.67,E2 -6917.67} C_VEL
LIN {X 0,Y 482.229,Z 361.989,A -85,B 0,C 180,E1 -6918.653,E2 -6918.653} C_VEL
LIN {X 0,Y 481.759,Z 371.163,A -85,B 0,C 180,E1 -6919.705,E2 -6919.705} C_VEL
LIN {X 0,Y 481.415,Z 380.106,A -85,B 0,C 180,E1 -6920.971,E2 -6920.971} C_VEL
LIN {X 0,Y 481.152,Z 387.304,A -85,B 0,C 180,E1 -6922.235,E2 -6922.235} C_VEL
LIN {X 0,Y 481.003,Z 393.032,A -85,B 0,C 180,E1 -6923.494,E2 -6923.494} C_VEL
LIN {X 0,Y 480.897,Z 398.198,A -85,B 0,C 180,E1 -6924.969,E2 -6924.969} C_VEL
LIN {X 0,Y 480.828,Z 400.494,A -85,B 0,C 180,E1 -6925.809,E2 -6925.809} C_VEL
LIN {X 0,Y 480.888,Z 402.357,A -85,B 0,C 180,E1 -6926.649,E2 -6926.649} C_VEL
LIN {X 0,Y 480.792,Z 404.747,A -85,B 0,C 180,E1 -6928.325,E2 -6928.325} C_VEL
LIN {X 0,Y 480.76,Z 405.355,A -85,B 0,C 180,E1 -6929.162,E2 -6929.162} C_VEL
LIN {X 0,Y 480.743,Z 405.571,A -85,B 0,C 180,E1 -6930,E2 -6930} C_VEL
LIN {X 0,Y 480.792,Z 404.749,A -85,B 0,C 180,E1 -6931.675,E2 -6931.675} C_VEL
LIN {X 0,Y 480.888,Z 402.361,A -85,B 0,C 180,E1 -6933.351,E2 -6933.351} C_VEL
LIN {X 0,Y 480.839,Z 399.424,A -85,B 0,C 180,E1 -6934.611,E2 -6934.611} C_VEL
LIN {X 0,Y 480.93,Z 395.452,A -85,B 0,C 180,E1 -6935.871,E2 -6935.871} C_VEL
LIN {X 0,Y 481.111,Z 389.344,A -85,B 0,C 180,E1 -6937.343,E2 -6937.343} C_VEL
LIN {X 0,Y 481.324,Z 382.668,A -85,B 0,C 180,E1 -6938.607,E2 -6938.607} C_VEL
LIN {X 0,Y 481.644,Z 374.385,A -85,B 0,C 180,E1 -6939.872,E2 -6939.872} C_VEL
LIN {X 0,Y 482.018,Z 365.897,A -85,B 0,C 180,E1 -6940.926,E2 -6940.926} C_VEL
LIN {X 0,Y 482.438,Z 355.43,A -85,B 0,C 180,E1 -6941.979,E2 -6941.979} C_VEL
LIN {X 0,Y 482.847,Z 344.321,A -85,B 0,C 180,E1 -6942.878,E2 -6942.878} C_VEL
LIN {X 0,Y 483.289,Z 333.658,A -85,B 0,C 180,E1 -6943.562,E2 -6943.562} C_VEL
LIN {X 0,Y 483.717,Z 321.994,A -85,B 0,C 180,E1 -6944.139,E2 -6944.139} C_VEL
LIN {X 0,Y 483.667,Z 315.561,A -85,B 0,C 180,E1 -6944.395,E2 -6944.395} C_VEL
LIN {X 0,Y 481.661,Z 302.494,A -85,B 0,C 180,E1 -6944.841,E2 -6944.841} C_VEL
LIN {X 0,Y 481.079,Z 298.823,A -85,B 0,C 180,E1 -6944.948,E2 -6944.948} C_VEL
LIN {X 0,Y 481.219,Z 291.52,A -85,B 0,C 180,E1 -6947.86,E2 -6947.86} C_VEL
LIN {X 0,Y 481.437,Z 283.959,A -85,B 0,C 180,E1 -6950.889,E2 -6950.889} C_VEL
LIN {X 0,Y 481.591,Z 275.979,A -85,B 0,C 180,E1 -6954.118,E2 -6954.118} C_VEL
LIN {X 0,Y 481.795,Z 268.662,A -85,B 0,C 180,E1 -6957.15,E2 -6957.15} C_VEL
LIN {X 0,Y 482.136,Z 261.539,A -85,B 0,C 180,E1 -6960.192,E2 -6960.192} C_VEL
LIN {X 0,Y 482.356,Z 254.91,A -85,B 0,C 180,E1 -6963.119,E2 -6963.119} C_VEL
LIN {X 0,Y 482.531,Z 249.446,A -85,B 0,C 180,E1 -6965.633,E2 -6965.633} C_VEL
LIN {X 0,Y 481.862,Z 244.548,A -85,B 0,C 180,E1 -6968.038,E2 -6968.038} C_VEL
LIN {X 0,Y 481.7,Z 243.485,A -85,B 0,C 180,E1 -6968.633,E2 -6968.633} C_VEL
LIN {X 0,Y 481.655,Z 243.492,A -85,B 0,C 180,E1 -6971.913,E2 -6971.913} C_VEL
LIN {X 0,Y 481.656,Z 243.488,A -85,B 0,C 180,E1 -6974.458,E2 -6974.458} C_VEL
LIN {X 0,Y 481.63,Z 243.49,A -85,B 0,C 180,E1 -6977.837,E2 -6977.837} C_VEL
LIN {X 0,Y 481.666,Z 243.485,A -85,B 0,C 180,E1 -6981.14,E2 -6981.14} C_VEL
LIN {X 0,Y 481.662,Z 243.486,A -85,B 0,C 180,E1 -6984.796,E2 -6984.796} C_VEL
LIN {X 0,Y 481.674,Z 243.486,A -85,B 0,C 180,E1 -6987.326,E2 -6987.326} C_VEL
LIN {X 0,Y 481.675,Z 243.486,A -85,B 0,C 180,E1 -6990.259,E2 -6990.259} C_VEL
LIN {X 0,Y 481.663,Z 243.486,A -85,B 0,C 180,E1 -6993.107,E2 -6993.107} C_VEL
LIN {X 0,Y 481.65,Z 243.491,A -85,B 0,C 180,E1 -6995.885,E2 -6995.885} C_VEL
LIN {X 0,Y 481.705,Z 243.481,A -85,B 0,C 180,E1 -6999.028,E2 -6999.028} C_VEL
LIN {X 0,Y 481.706,Z 243.482,A -85,B 0,C 180,E1 -7002.158,E2 -7002.158} C_VEL
LIN {X 0,Y 481.744,Z 243.477,A -85,B 0,C 180,E1 -7004.776,E2 -7004.776} C_VEL
LIN {X 0,Y 481.751,Z 243.476,A -85,B 0,C 180,E1 -7008.215,E2 -7008.215} C_VEL
LIN {X 0,Y 481.738,Z 243.48,A -85,B 0,C 180,E1 -7011.611,E2 -7011.611} C_VEL
LIN {X 0,Y 481.809,Z 243.468,A -85,B 0,C 180,E1 -7014.14,E2 -7014.14} C_VEL
LIN {X 0,Y 481.93,Z 243.454,A -85,B 0,C 180,E1 -7017.493,E2 -7017.493} C_VEL
LIN {X 0,Y 481.941,Z 243.453,A -85,B 0,C 180,E1 -7020,E2 -7020} C_VEL
LIN {X 0,Y 481.915,Z 243.454,A -85,B 0,C 180,E1 -7022.508,E2 -7022.508} C_VEL
LIN {X 0,Y 481.797,Z 243.467,A -85,B 0,C 180,E1 -7025.861,E2 -7025.861} C_VEL
LIN {X 0,Y 481.743,Z 243.477,A -85,B 0,C 180,E1 -7028.389,E2 -7028.389} C_VEL
LIN {X 0,Y 481.753,Z 243.476,A -85,B 0,C 180,E1 -7031.785,E2 -7031.785} C_VEL
LIN {X 0,Y 481.744,Z 243.479,A -85,B 0,C 180,E1 -7035.224,E2 -7035.224} C_VEL
LIN {X 0,Y 481.709,Z 243.485,A -85,B 0,C 180,E1 -7038.722,E2 -7038.722} C_VEL
LIN {X 0,Y 481.648,Z 243.486,A -85,B 0,C 180,E1 -7041.395,E2 -7041.395} C_VEL
LIN {X 0,Y 481.663,Z 243.49,A -85,B 0,C 180,E1 -7044.114,E2 -7044.114} C_VEL
LIN {X 0,Y 481.748,Z 243.477,A -85,B 0,C 180,E1 -7047.139,E2 -7047.139} C_VEL
LIN {X 0,Y 481.679,Z 243.485,A -85,B 0,C 180,E1 -7049.741,E2 -7049.741} C_VEL
LIN {X 0,Y 481.654,Z 243.489,A -85,B 0,C 180,E1 -7052.676,E2 -7052.676} C_VEL
LIN {X 0,Y 481.632,Z 243.491,A -85,B 0,C 180,E1 -7055.71,E2 -7055.71} C_VEL
LIN {X 0,Y 481.672,Z 243.485,A -85,B 0,C 180,E1 -7058.859,E2 -7058.859} C_VEL
LIN {X 0,Y 481.648,Z 243.489,A -85,B 0,C 180,E1 -7061.912,E2 -7061.912} C_VEL
LIN {X 0,Y 481.655,Z 243.489,A -85,B 0,C 180,E1 -7064.458,E2 -7064.458} C_VEL
LIN {X 0,Y 481.615,Z 243.497,A -85,B 0,C 180,E1 -7067.836,E2 -7067.836} C_VEL
LIN {X 0,Y 481.669,Z 243.486,A -85,B 0,C 180,E1 -7071.141,E2 -7071.141} C_VEL
LIN {X 0,Y 481.543,Z 243.503,A -85,B 0,C 180,E1 -7074.282,E2 -7074.282} C_VEL
LIN {X 0,Y 481.531,Z 243.74,A -85,B 0,C 180,E1 -7074.818,E2 -7074.818} C_VEL
LIN {X 0,Y 481.512,Z 247.218,A -85,B 0,C 180,E1 -7077.314,E2 -7077.314} C_VEL
LIN {X 0,Y 481.403,Z 251.391,A -85,B 0,C 180,E1 -7080.24,E2 -7080.24} C_VEL
LIN {X 0,Y 481.277,Z 255.543,A -85,B 0,C 180,E1 -7083.084,E2 -7083.084} C_VEL
LIN {X 0,Y 481.224,Z 259.674,A -85,B 0,C 180,E1 -7085.863,E2 -7085.863} C_VEL
LIN {X 0,Y 481.14,Z 262.476,A -85,B 0,C 180,E1 -7087.713,E2 -7087.713} C_VEL
LIN {X 0,Y 480.421,Z 263.592,A -85,B 0,C 180,E1 -7088.399,E2 -7088.399} C_VEL
LIN {X 0,Y 477.516,Z 265.577,A -85,B 0,C 180,E1 -7089.509,E2 -7089.509} C_VEL
LIN {X 0,Y 475.087,Z 267.187,A -85,B 0,C 180,E1 -7090.403,E2 -7090.403} C_VEL
LIN {X 0,Y 474.05,Z 268.357,A -85,B 0,C 180,E1 -7091.095,E2 -7091.095} C_VEL
LIN {X 0,Y 473.967,Z 268.731,A -85,B 0,C 180,E1 -7091.33,E2 -7091.33} C_VEL
LIN {X 0,Y 473.994,Z 274.48,A -85,B 0,C 180,E1 -7094.91,E2 -7094.91} C_VEL
LIN {X 0,Y 476.61,Z 287.761,A -85,B 0,C 180,E1 -7095.373,E2 -7095.373} C_VEL
LIN {X 0,Y 477.135,Z 292.109,A -85,B 0,C 180,E1 -7095.553,E2 -7095.553} C_VEL
LIN {X 0,Y 476.707,Z 304.665,A -85,B 0,C 180,E1 -7096.139,E2 -7096.139} C_VEL
LIN {X 0,Y 476.294,Z 316.499,A -85,B 0,C 180,E1 -7096.874,E2 -7096.874} C_VEL
LIN {X 0,Y 475.856,Z 327.376,A -85,B 0,C 180,E1 -7097.742,E2 -7097.742} C_VEL
LIN {X 0,Y 475.414,Z 337.105,A -85,B 0,C 180,E1 -7098.704,E2 -7098.704} C_VEL
LIN {X 0,Y 474.99,Z 345.954,A -85,B 0,C 180,E1 -7099.773,E2 -7099.773} C_VEL
LIN {X 0,Y 474.571,Z 354.587,A -85,B 0,C 180,E1 -7101.054,E2 -7101.054} C_VEL
LIN {X 0,Y 474.234,Z 361.468,A -85,B 0,C 180,E1 -7102.335,E2 -7102.335} C_VEL
LIN {X 0,Y 474.103,Z 366.881,A -85,B 0,C 180,E1 -7103.592,E2 -7103.592} C_VEL
LIN {X 0,Y 473.855,Z 371.302,A -85,B 0,C 180,E1 -7104.895,E2 -7104.895} C_VEL
LIN {X 0,Y 473.872,Z 373.588,A -85,B 0,C 180,E1 -7105.747,E2 -7105.747} C_VEL
LIN {X 0,Y 473.842,Z 375.45,A -85,B 0,C 180,E1 -7106.599,E2 -7106.599} C_VEL
LIN {X 0,Y 473.763,Z 376.856,A -85,B 0,C 180,E1 -7107.449,E2 -7107.449} C_VEL
LIN {X 0,Y 473.689,Z 378.47,A -85,B 0,C 180,E1 -7109.15,E2 -7109.15} C_VEL
LIN {X 0,Y 473.67,Z 378.706,A -85,B 0,C 180,E1 -7110,E2 -7110} C_VEL
LIN {X 0,Y 473.689,Z 378.52,A -85,B 0,C 180,E1 -7110.85,E2 -7110.85} C_VEL
LIN {X 0,Y 473.763,Z 376.971,A -85,B 0,C 180,E1 -7112.551,E2 -7112.551} C_VEL
LIN {X 0,Y 473.841,Z 375.615,A -85,B 0,C 180,E1 -7113.401,E2 -7113.401} C_VEL
LIN {X 0,Y 473.823,Z 372.755,A -85,B 0,C 180,E1 -7114.679,E2 -7114.679} C_VEL
LIN {X 0,Y 474.086,Z 368.868,A -85,B 0,C 180,E1 -7115.956,E2 -7115.956} C_VEL
LIN {X 0,Y 474.148,Z 363.861,A -85,B 0,C 180,E1 -7117.238,E2 -7117.238} C_VEL
LIN {X 0,Y 474.417,Z 357.555,A -85,B 0,C 180,E1 -7118.519,E2 -7118.519} C_VEL
LIN {X 0,Y 474.776,Z 349.658,A -85,B 0,C 180,E1 -7119.801,E2 -7119.801} C_VEL
LIN {X 0,Y 475.155,Z 341.608,A -85,B 0,C 180,E1 -7120.87,E2 -7120.87} C_VEL
LIN {X 0,Y 475.632,Z 331.783,A -85,B 0,C 180,E1 -7121.939,E2 -7121.939} C_VEL
LIN {X 0,Y 476.107,Z 320.906,A -85,B 0,C 180,E1 -7122.888,E2 -7122.888} C_VEL
LIN {X 0,Y 476.541,Z 309.906,A -85,B 0,C 180,E1 -7123.649,E2 -7123.649} C_VEL
LIN {X 0,Y 476.969,Z 297.944,A -85,B 0,C 180,E1 -7124.289,E2 -7124.289} C_VEL
LIN {X 0,Y 476.903,Z 289.248,A -85,B 0,C 180,E1 -7124.655,E2 -7124.655} C_VEL
LIN {X 0,Y 474.28,Z 276.142,A -85,B 0,C 180,E1 -7125.132,E2 -7125.132} C_VEL
LIN {X 0,Y 473.978,Z 274.429,A -85,B 0,C 180,E1 -7125.204,E2 -7125.204} C_VEL
LIN {X 0,Y 473.982,Z 268.302,A -85,B 0,C 180,E1 -7129.039,E2 -7129.039} C_VEL
LIN {X 0,Y 474.064,Z 264.091,A -85,B 0,C 180,E1 -7131.754,E2 -7131.754} C_VEL
LIN {X 0,Y 474.136,Z 259.968,A -85,B 0,C 180,E1 -7134.522,E2 -7134.522} C_VEL
LIN {X 0,Y 474.24,Z 255.818,A -85,B 0,C 180,E1 -7137.349,E2 -7137.349} C_VEL
LIN {X 0,Y 474.346,Z 251.642,A -85,B 0,C 180,E1 -7140.249,E2 -7140.249} C_VEL
LIN {X 0,Y 474.447,Z 247.448,A -85,B 0,C 180,E1 -7143.236,E2 -7143.236} C_VEL
LIN {X 0,Y 474.469,Z 244.418,A -85,B 0,C 180,E1 -7145.444,E2 -7145.444} C_VEL
LIN {X 0,Y 474.612,Z 244.367,A -85,B 0,C 180,E1 -7148.458,E2 -7148.458} C_VEL
LIN {X 0,Y 474.597,Z 244.366,A -85,B 0,C 180,E1 -7151.788,E2 -7151.788} C_VEL
LIN {X 0,Y 474.616,Z 244.365,A -85,B 0,C 180,E1 -7154.702,E2 -7154.702} C_VEL
LIN {X 0,Y 474.618,Z 244.365,A -85,B 0,C 180,E1 -7158.214,E2 -7158.214} C_VEL
LIN {X 0,Y 474.614,Z 244.364,A -85,B 0,C 180,E1 -7161.543,E2 -7161.543} C_VEL
LIN {X 0,Y 474.625,Z 244.361,A -85,B 0,C 180,E1 -7164.726,E2 -7164.726} C_VEL
LIN {X 0,Y 474.637,Z 244.365,A -85,B 0,C 180,E1 -7167.788,E2 -7167.788} C_VEL
LIN {X 0,Y 474.624,Z 244.364,A -85,B 0,C 180,E1 -7170.885,E2 -7170.885} C_VEL
LIN {X 0,Y 474.657,Z 244.36,A -85,B 0,C 180,E1 -7173.628,E2 -7173.628} C_VEL
LIN {X 0,Y 474.638,Z 244.361,A -85,B 0,C 180,E1 -7176.642,E2 -7176.642} C_VEL
LIN {X 0,Y 474.654,Z 244.358,A -85,B 0,C 180,E1 -7180.089,E2 -7180.089} C_VEL
LIN {X 0,Y 474.627,Z 244.364,A -85,B 0,C 180,E1 -7182.773,E2 -7182.773} C_VEL
LIN {X 0,Y 474.646,Z 244.361,A -85,B 0,C 180,E1 -7185.421,E2 -7185.421} C_VEL
LIN {X 0,Y 474.708,Z 244.354,A -85,B 0,C 180,E1 -7188.038,E2 -7188.038} C_VEL
LIN {X 0,Y 474.716,Z 244.354,A -85,B 0,C 180,E1 -7191.486,E2 -7191.486} C_VEL
LIN {X 0,Y 474.762,Z 244.343,A -85,B 0,C 180,E1 -7194.052,E2 -7194.052} C_VEL
LIN {X 0,Y 474.882,Z 244.331,A -85,B 0,C 180,E1 -7197.455,E2 -7197.455} C_VEL
LIN {X 0,Y 474.886,Z 244.332,A -85,B 0,C 180,E1 -7200,E2 -7200} C_VEL
LIN {X 0,Y 474.897,Z 244.33,A -85,B 0,C 180,E1 -7202.545,E2 -7202.545} C_VEL
LIN {X 0,Y 474.773,Z 244.344,A -85,B 0,C 180,E1 -7205.948,E2 -7205.948} C_VEL
LIN {X 0,Y 474.705,Z 244.357,A -85,B 0,C 180,E1 -7208.514,E2 -7208.514} C_VEL
LIN {X 0,Y 474.695,Z 244.356,A -85,B 0,C 180,E1 -7211.963,E2 -7211.963} C_VEL
LIN {X 0,Y 474.703,Z 244.354,A -85,B 0,C 180,E1 -7215.456,E2 -7215.456} C_VEL
LIN {X 0,Y 474.668,Z 244.358,A -85,B 0,C 180,E1 -7219.01,E2 -7219.01} C_VEL
LIN {X 0,Y 474.591,Z 244.367,A -85,B 0,C 180,E1 -7221.729,E2 -7221.729} C_VEL
LIN {X 0,Y 474.629,Z 244.361,A -85,B 0,C 180,E1 -7224.495,E2 -7224.495} C_VEL
LIN {X 0,Y 474.639,Z 244.362,A -85,B 0,C 180,E1 -7227.324,E2 -7227.324} C_VEL
LIN {X 0,Y 474.604,Z 244.367,A -85,B 0,C 180,E1 -7230.23,E2 -7230.23} C_VEL
LIN {X 0,Y 474.646,Z 244.361,A -85,B 0,C 180,E1 -7233.22,E2 -7233.22} C_VEL
LIN {X 0,Y 474.586,Z 244.368,A -85,B 0,C 180,E1 -7236.324,E2 -7236.324} C_VEL
LIN {X 0,Y 474.623,Z 244.366,A -85,B 0,C 180,E1 -7239.548,E2 -7239.548} C_VEL
LIN {X 0,Y 474.59,Z 244.367,A -85,B 0,C 180,E1 -7242.232,E2 -7242.232} C_VEL
LIN {X 0,Y 474.619,Z 244.364,A -85,B 0,C 180,E1 -7245.298,E2 -7245.298} C_VEL
LIN {X 0,Y 474.623,Z 244.368,A -85,B 0,C 180,E1 -7248.215,E2 -7248.215} C_VEL
LIN {X 0,Y 474.675,Z 244.505,A -85,B 0,C 180,E1 -7251.277,E2 -7251.277} C_VEL
LIN {X 0,Y 475.419,Z 249.389,A -85,B 0,C 180,E1 -7253.75,E2 -7253.75} C_VEL
LIN {X 0,Y 475.476,Z 253.843,A -85,B 0,C 180,E1 -7255.867,E2 -7255.867} C_VEL
LIN {X 0,Y 475.163,Z 260.348,A -85,B 0,C 180,E1 -7258.823,E2 -7258.823} C_VEL
LIN {X 0,Y 474.847,Z 266.98,A -85,B 0,C 180,E1 -7261.73,E2 -7261.73} C_VEL
LIN {X 0,Y 474.626,Z 274.761,A -85,B 0,C 180,E1 -7265.044,E2 -7265.044} C_VEL
LIN {X 0,Y 474.415,Z 282.546,A -85,B 0,C 180,E1 -7268.263,E2 -7268.263} C_VEL
LIN {X 0,Y 474.18,Z 290.567,A -85,B 0,C 180,E1 -7271.545,E2 -7271.545} C_VEL
LIN {X 0,Y 474.035,Z 298.789,A -85,B 0,C 180,E1 -7274.838,E2 -7274.838} C_VEL
LIN {X 0,Y 476.154,Z 311.93,A -85,B 0,C 180,E1 -7275.249,E2 -7275.249} C_VEL
LIN {X 0,Y 476.869,Z 319.21,A -85,B 0,C 180,E1 -7275.545,E2 -7275.545} C_VEL
LIN {X 0,Y 476.41,Z 331.545,A -85,B 0,C 180,E1 -7276.13,E2 -7276.13} C_VEL
LIN {X 0,Y 475.951,Z 343.409,A -85,B 0,C 180,E1 -7276.878,E2 -7276.878} C_VEL
LIN {X 0,Y 475.516,Z 353.536,A -85,B 0,C 180,E1 -7277.688,E2 -7277.688} C_VEL
LIN {X 0,Y 475.116,Z 363.748,A -85,B 0,C 180,E1 -7278.697,E2 -7278.697} C_VEL
LIN {X 0,Y 474.643,Z 372.597,A -85,B 0,C 180,E1 -7279.765,E2 -7279.765} C_VEL
LIN {X 0,Y 474.313,Z 381.23,A -85,B 0,C 180,E1 -7281.049,E2 -7281.049} C_VEL
LIN {X 0,Y 474.044,Z 388.13,A -85,B 0,C 180,E1 -7282.332,E2 -7282.332} C_VEL
LIN {X 0,Y 473.905,Z 393.304,A -85,B 0,C 180,E1 -7283.52,E2 -7283.52} C_VEL
LIN {X 0,Y 473.828,Z 397.999,A -85,B 0,C 180,E1 -7284.894,E2 -7284.894} C_VEL
LIN {X 0,Y 473.734,Z 400.294,A -85,B 0,C 180,E1 -7285.746,E2 -7285.746} C_VEL
LIN {X 0,Y 473.795,Z 402.158,A -85,B 0,C 180,E1 -7286.598,E2 -7286.598} C_VEL
LIN {X 0,Y 473.741,Z 403.552,A -85,B 0,C 180,E1 -7287.449,E2 -7287.449} C_VEL
LIN {X 0,Y 473.688,Z 405.156,A -85,B 0,C 180,E1 -7289.15,E2 -7289.15} C_VEL
LIN {X 0,Y 473.669,Z 405.372,A -85,B 0,C 180,E1 -7290,E2 -7290} C_VEL
LIN {X 0,Y 473.688,Z 405.156,A -85,B 0,C 180,E1 -7290.85,E2 -7290.85} C_VEL
LIN {X 0,Y 473.741,Z 403.555,A -85,B 0,C 180,E1 -7292.551,E2 -7292.551} C_VEL
LIN {X 0,Y 473.795,Z 402.161,A -85,B 0,C 180,E1 -7293.401,E2 -7293.401} C_VEL
LIN {X 0,Y 473.762,Z 399.224,A -85,B 0,C 180,E1 -7294.68,E2 -7294.68} C_VEL
LIN {X 0,Y 473.838,Z 395.251,A -85,B 0,C 180,E1 -7295.959,E2 -7295.959} C_VEL
LIN {X 0,Y 474.029,Z 389.142,A -85,B 0,C 180,E1 -7297.454,E2 -7297.454} C_VEL
LIN {X 0,Y 474.287,Z 382.466,A -85,B 0,C 180,E1 -7298.736,E2 -7298.736} C_VEL
LIN {X 0,Y 474.594,Z 374.182,A -85,B 0,C 180,E1 -7300.02,E2 -7300.02} C_VEL
LIN {X 0,Y 475.023,Z 365.695,A -85,B 0,C 180,E1 -7301.089,E2 -7301.089} C_VEL
LIN {X 0,Y 475.445,Z 355.428,A -85,B 0,C 180,E1 -7302.139,E2 -7302.139} C_VEL
LIN {X 0,Y 475.923,Z 343.829,A -85,B 0,C 180,E1 -7303.09,E2 -7303.09} C_VEL
LIN {X 0,Y 476.422,Z 331.53,A -85,B 0,C 180,E1 -7303.87,E2 -7303.87} C_VEL
LIN {X 0,Y 476.868,Z 319.183,A -85,B 0,C 180,E1 -7304.455,E2 -7304.455} C_VEL
LIN {X 0,Y 475.802,Z 309.678,A -85,B 0,C 180,E1 -7304.83,E2 -7304.83} C_VEL
LIN {X 0,Y 474.007,Z 298.633,A -85,B 0,C 180,E1 -7305.176,E2 -7305.176} C_VEL
LIN {X 0,Y 474.18,Z 290.563,A -85,B 0,C 180,E1 -7308.455,E2 -7308.455} C_VEL
LIN {X 0,Y 474.414,Z 282.543,A -85,B 0,C 180,E1 -7311.737,E2 -7311.737} C_VEL
LIN {X 0,Y 474.629,Z 274.748,A -85,B 0,C 180,E1 -7314.956,E2 -7314.956} C_VEL
LIN {X 0,Y 474.841,Z 266.959,A -85,B 0,C 180,E1 -7318.27,E2 -7318.27} C_VEL
LIN {X 0,Y 475.132,Z 260.918,A -85,B 0,C 180,E1 -7320.916,E2 -7320.916} C_VEL
LIN {X 0,Y 475.432,Z 254.867,A -85,B 0,C 180,E1 -7323.646,E2 -7323.646} C_VEL
LIN {X 0,Y 475.524,Z 250.654,A -85,B 0,C 180,E1 -7325.622,E2 -7325.622} C_VEL
LIN {X 0,Y 475.102,Z 247.192,A -85,B 0,C 180,E1 -7327.337,E2 -7327.337} C_VEL
LIN {X 0,Y 474.665,Z 244.361,A -85,B 0,C 180,E1 -7328.86,E2 -7328.86} C_VEL
LIN {X 0,Y 474.626,Z 244.369,A -85,B 0,C 180,E1 -7332.237,E2 -7332.237} C_VEL
LIN {X 0,Y 474.617,Z 244.368,A -85,B 0,C 180,E1 -7335.298,E2 -7335.298} C_VEL
LIN {X 0,Y 474.604,Z 244.365,A -85,B 0,C 180,E1 -7338.213,E2 -7338.213} C_VEL
LIN {X 0,Y 474.608,Z 244.363,A -85,B 0,C 180,E1 -7341.542,E2 -7341.542} C_VEL
LIN {X 0,Y 474.624,Z 244.363,A -85,B 0,C 180,E1 -7344.725,E2 -7344.725} C_VEL
LIN {X 0,Y 474.638,Z 244.364,A -85,B 0,C 180,E1 -7347.788,E2 -7347.788} C_VEL
LIN {X 0,Y 474.608,Z 244.367,A -85,B 0,C 180,E1 -7350.888,E2 -7350.888} C_VEL
LIN {X 0,Y 474.592,Z 244.366,A -85,B 0,C 180,E1 -7353.624,E2 -7353.624} C_VEL
LIN {X 0,Y 474.635,Z 244.36,A -85,B 0,C 180,E1 -7356.642,E2 -7356.642} C_VEL
LIN {X 0,Y 474.657,Z 244.36,A -85,B 0,C 180,E1 -7360.09,E2 -7360.09} C_VEL
LIN {X 0,Y 474.65,Z 244.361,A -85,B 0,C 180,E1 -7362.774,E2 -7362.774} C_VEL
LIN {X 0,Y 474.646,Z 244.361,A -85,B 0,C 180,E1 -7365.421,E2 -7365.421} C_VEL
LIN {X 0,Y 474.705,Z 244.355,A -85,B 0,C 180,E1 -7368.038,E2 -7368.038} C_VEL
LIN {X 0,Y 474.71,Z 244.357,A -85,B 0,C 180,E1 -7371.486,E2 -7371.486} C_VEL
LIN {X 0,Y 474.772,Z 244.344,A -85,B 0,C 180,E1 -7374.052,E2 -7374.052} C_VEL
LIN {X 0,Y 474.896,Z 244.33,A -85,B 0,C 180,E1 -7377.455,E2 -7377.455} C_VEL
LIN {X 0,Y 474.911,Z 244.329,A -85,B 0,C 180,E1 -7380,E2 -7380} C_VEL
LIN {X 0,Y 474.881,Z 244.331,A -85,B 0,C 180,E1 -7382.545,E2 -7382.545} C_VEL
LIN {X 0,Y 474.76,Z 244.344,A -85,B 0,C 180,E1 -7385.948,E2 -7385.948} C_VEL
LIN {X 0,Y 474.715,Z 244.354,A -85,B 0,C 180,E1 -7388.514,E2 -7388.514} C_VEL
LIN {X 0,Y 474.707,Z 244.354,A -85,B 0,C 180,E1 -7391.962,E2 -7391.962} C_VEL
LIN {X 0,Y 474.701,Z 244.355,A -85,B 0,C 180,E1 -7395.456,E2 -7395.456} C_VEL
LIN {X 0,Y 474.663,Z 244.359,A -85,B 0,C 180,E1 -7399.01,E2 -7399.01} C_VEL
LIN {X 0,Y 474.591,Z 244.366,A -85,B 0,C 180,E1 -7401.729,E2 -7401.729} C_VEL
LIN {X 0,Y 474.643,Z 244.362,A -85,B 0,C 180,E1 -7404.494,E2 -7404.494} C_VEL
LIN {X 0,Y 474.682,Z 244.357,A -85,B 0,C 180,E1 -7407.334,E2 -7407.334} C_VEL
LIN {X 0,Y 474.604,Z 244.367,A -85,B 0,C 180,E1 -7410.81,E2 -7410.81} C_VEL
LIN {X 0,Y 474.622,Z 244.365,A -85,B 0,C 180,E1 -7413.981,E2 -7413.981} C_VEL
LIN {X 0,Y 474.568,Z 244.368,A -85,B 0,C 180,E1 -7416.898,E2 -7416.898} C_VEL
LIN {X 0,Y 474.615,Z 244.368,A -85,B 0,C 180,E1 -7419.646,E2 -7419.646} C_VEL
LIN {X 0,Y 474.602,Z 244.367,A -85,B 0,C 180,E1 -7422.234,E2 -7422.234} C_VEL
LIN {X 0,Y 474.615,Z 244.365,A -85,B 0,C 180,E1 -7425.298,E2 -7425.298} C_VEL
LIN {X 0,Y 474.592,Z 244.367,A -85,B 0,C 180,E1 -7428.211,E2 -7428.211} C_VEL
LIN {X 0,Y 474.61,Z 244.368,A -85,B 0,C 180,E1 -7431.542,E2 -7431.542} C_VEL
LIN {X 0,Y 474.485,Z 244.384,A -85,B 0,C 180,E1 -7434.553,E2 -7434.553} C_VEL
LIN {X 0,Y 474.474,Z 247.315,A -85,B 0,C 180,E1 -7436.767,E2 -7436.767} C_VEL
LIN {X 0,Y 474.364,Z 251.502,A -85,B 0,C 180,E1 -7439.753,E2 -7439.753} C_VEL
LIN {X 0,Y 474.235,Z 255.842,A -85,B 0,C 180,E1 -7442.771,E2 -7442.771} C_VEL
LIN {X 0,Y 474.153,Z 259.813,A -85,B 0,C 180,E1 -7445.479,E2 -7445.479} C_VEL
LIN {X 0,Y 474.062,Z 263.95,A -85,B 0,C 180,E1 -7448.246,E2 -7448.246} C_VEL
LIN {X 0,Y 473.967,Z 268.731,A -85,B 0,C 180,E1 -7451.33,E2 -7451.33} C_VEL
LIN {X 0,Y 473.277,Z 269.517,A -85,B 0,C 180,E1 -7451.793,E2 -7451.793} C_VEL
LIN {X 0,Y 470.382,Z 270.903,A -85,B 0,C 180,E1 -7452.512,E2 -7452.512} C_VEL
LIN {X 0,Y 467.491,Z 272.301,A -85,B 0,C 180,E1 -7453.239,E2 -7453.239} C_VEL
LIN {X 0,Y 466.827,Z 273.108,A -85,B 0,C 180,E1 -7453.712,E2 -7453.712} C_VEL
LIN {X 0,Y 466.925,Z 274.619,A -85,B 0,C 180,E1 -7454.658,E2 -7454.658} C_VEL
LIN {X 0,Y 470.021,Z 290.359,A -85,B 0,C 180,E1 -7455.251,E2 -7455.251} C_VEL
LIN {X 0,Y 470.204,Z 294.916,A -85,B 0,C 180,E1 -7455.446,E2 -7455.446} C_VEL
LIN {X 0,Y 469.774,Z 306.85,A -85,B 0,C 180,E1 -7456.041,E2 -7456.041} C_VEL
LIN {X 0,Y 469.348,Z 317.472,A -85,B 0,C 180,E1 -7456.733,E2 -7456.733} C_VEL
LIN {X 0,Y 468.851,Z 328.751,A -85,B 0,C 180,E1 -7457.666,E2 -7457.666} C_VEL
LIN {X 0,Y 468.3,Z 339.254,A -85,B 0,C 180,E1 -7458.75,E2 -7458.75} C_VEL
LIN {X 0,Y 467.905,Z 347.758,A -85,B 0,C 180,E1 -7459.835,E2 -7459.835} C_VEL
LIN {X 0,Y 467.485,Z 356.018,A -85,B 0,C 180,E1 -7461.136,E2 -7461.136} C_VEL
LIN {X 0,Y 467.149,Z 362.672,A -85,B 0,C 180,E1 -7462.436,E2 -7462.436} C_VEL
LIN {X 0,Y 467.016,Z 368.765,A -85,B 0,C 180,E1 -7463.953,E2 -7463.953} C_VEL
LIN {X 0,Y 466.75,Z 372.728,A -85,B 0,C 180,E1 -7465.25,E2 -7465.25} C_VEL
LIN {X 0,Y 466.774,Z 375.65,A -85,B 0,C 180,E1 -7466.547,E2 -7466.547} C_VEL
LIN {X 0,Y 466.683,Z 377.056,A -85,B 0,C 180,E1 -7467.411,E2 -7467.411} C_VEL
LIN {X 0,Y 466.62,Z 378.67,A -85,B 0,C 180,E1 -7469.137,E2 -7469.137} C_VEL
LIN {X 0,Y 466.599,Z 378.906,A -85,B 0,C 180,E1 -7470,E2 -7470} C_VEL
LIN {X 0,Y 466.619,Z 378.719,A -85,B 0,C 180,E1 -7470.863,E2 -7470.863} C_VEL
LIN {X 0,Y 466.683,Z 377.17,A -85,B 0,C 180,E1 -7472.59,E2 -7472.59} C_VEL
LIN {X 0,Y 466.773,Z 375.814,A -85,B 0,C 180,E1 -7473.453,E2 -7473.453} C_VEL
LIN {X 0,Y 466.743,Z 372.954,A -85,B 0,C 180,E1 -7474.751,E2 -7474.751} C_VEL
LIN {X 0,Y 467.01,Z 369.066,A -85,B 0,C 180,E1 -7476.047,E2 -7476.047} C_VEL
LIN {X 0,Y 467.102,Z 364.059,A -85,B 0,C 180,E1 -7477.348,E2 -7477.348} C_VEL
LIN {X 0,Y 467.379,Z 357.753,A -85,B 0,C 180,E1 -7478.649,E2 -7478.649} C_VEL
LIN {X 0,Y 467.773,Z 349.855,A -85,B 0,C 180,E1 -7479.95,E2 -7479.95} C_VEL
LIN {X 0,Y 468.185,Z 341.804,A -85,B 0,C 180,E1 -7481.034,E2 -7481.034} C_VEL
LIN {X 0,Y 468.693,Z 331.978,A -85,B 0,C 180,E1 -7482.118,E2 -7482.118} C_VEL
LIN {X 0,Y 469.196,Z 320.934,A -85,B 0,C 180,E1 -7483.094,E2 -7483.094} C_VEL
LIN {X 0,Y 469.637,Z 310.098,A -85,B 0,C 180,E1 -7483.853,E2 -7483.853} C_VEL
LIN {X 0,Y 470.113,Z 298.134,A -85,B 0,C 180,E1 -7484.502,E2 -7484.502} C_VEL
LIN {X 0,Y 470.077,Z 290.642,A -85,B 0,C 180,E1 -7484.829,E2 -7484.829} C_VEL
LIN {X 0,Y 467.67,Z 278.322,A -85,B 0,C 180,E1 -7485.302,E2 -7485.302} C_VEL
LIN {X 0,Y 466.926,Z 274.612,A -85,B 0,C 180,E1 -7485.438,E2 -7485.438} C_VEL
LIN {X 0,Y 466.916,Z 269.75,A -85,B 0,C 180,E1 -7488.508,E2 -7488.508} C_VEL
LIN {X 0,Y 466.983,Z 265.651,A -85,B 0,C 180,E1 -7491.174,E2 -7491.174} C_VEL
LIN {X 0,Y 467.061,Z 261.484,A -85,B 0,C 180,E1 -7493.971,E2 -7493.971} C_VEL
LIN {X 0,Y 467.151,Z 257.34,A -85,B 0,C 180,E1 -7496.829,E2 -7496.829} C_VEL
LIN {X 0,Y 467.274,Z 253.153,A -85,B 0,C 180,E1 -7499.758,E2 -7499.758} C_VEL
LIN {X 0,Y 467.38,Z 248.941,A -85,B 0,C 180,E1 -7502.775,E2 -7502.775} C_VEL
LIN {X 0,Y 467.42,Z 246.137,A -85,B 0,C 180,E1 -7504.845,E2 -7504.845} C_VEL
LIN {X 0,Y 467.468,Z 245.256,A -85,B 0,C 180,E1 -7505.897,E2 -7505.897} C_VEL
LIN {X 0,Y 467.56,Z 245.247,A -85,B 0,C 180,E1 -7508.59,E2 -7508.59} C_VEL
LIN {X 0,Y 467.562,Z 245.242,A -85,B 0,C 180,E1 -7511.405,E2 -7511.405} C_VEL
LIN {X 0,Y 467.566,Z 245.244,A -85,B 0,C 180,E1 -7515.052,E2 -7515.052} C_VEL
LIN {X 0,Y 467.576,Z 245.244,A -85,B 0,C 180,E1 -7518.597,E2 -7518.597} C_VEL
LIN {X 0,Y 467.563,Z 245.242,A -85,B 0,C 180,E1 -7521.409,E2 -7521.409} C_VEL
LIN {X 0,Y 467.562,Z 245.245,A -85,B 0,C 180,E1 -7524.261,E2 -7524.261} C_VEL
LIN {X 0,Y 467.582,Z 245.241,A -85,B 0,C 180,E1 -7527.321,E2 -7527.321} C_VEL
LIN {X 0,Y 467.569,Z 245.243,A -85,B 0,C 180,E1 -7530.668,E2 -7530.668} C_VEL
LIN {X 0,Y 467.616,Z 245.238,A -85,B 0,C 180,E1 -7533.2,E2 -7533.2} C_VEL
LIN {X 0,Y 467.594,Z 245.238,A -85,B 0,C 180,E1 -7536.469,E2 -7536.469} C_VEL
LIN {X 0,Y 467.624,Z 245.236,A -85,B 0,C 180,E1 -7539.777,E2 -7539.777} C_VEL
LIN {X 0,Y 467.59,Z 245.239,A -85,B 0,C 180,E1 -7542.506,E2 -7542.506} C_VEL
LIN {X 0,Y 467.605,Z 245.239,A -85,B 0,C 180,E1 -7545.196,E2 -7545.196} C_VEL
LIN {X 0,Y 467.66,Z 245.232,A -85,B 0,C 180,E1 -7547.855,E2 -7547.855} C_VEL
LIN {X 0,Y 467.674,Z 245.233,A -85,B 0,C 180,E1 -7551.357,E2 -7551.357} C_VEL
LIN {X 0,Y 467.727,Z 245.22,A -85,B 0,C 180,E1 -7553.962,E2 -7553.962} C_VEL
LIN {X 0,Y 467.823,Z 245.21,A -85,B 0,C 180,E1 -7557.417,E2 -7557.417} C_VEL
LIN {X 0,Y 467.855,Z 245.207,A -85,B 0,C 180,E1 -7560,E2 -7560} C_VEL
LIN {X 0,Y 467.862,Z 245.206,A -85,B 0,C 180,E1 -7562.583,E2 -7562.583} C_VEL
LIN {X 0,Y 467.737,Z 245.221,A -85,B 0,C 180,E1 -7566.037,E2 -7566.037} C_VEL
LIN {X 0,Y 467.662,Z 245.234,A -85,B 0,C 180,E1 -7568.643,E2 -7568.643} C_VEL
LIN {X 0,Y 467.65,Z 245.234,A -85,B 0,C 180,E1 -7572.354,E2 -7572.354} C_VEL
LIN {X 0,Y 467.653,Z 245.234,A -85,B 0,C 180,E1 -7575.885,E2 -7575.885} C_VEL
LIN {X 0,Y 467.627,Z 245.236,A -85,B 0,C 180,E1 -7579.308,E2 -7579.308} C_VEL
LIN {X 0,Y 467.537,Z 245.249,A -85,B 0,C 180,E1 -7582.074,E2 -7582.074} C_VEL
LIN {X 0,Y 467.562,Z 245.24,A -85,B 0,C 180,E1 -7584.89,E2 -7584.89} C_VEL
LIN {X 0,Y 467.581,Z 245.243,A -85,B 0,C 180,E1 -7587.772,E2 -7587.772} C_VEL
LIN {X 0,Y 467.57,Z 245.243,A -85,B 0,C 180,E1 -7591.045,E2 -7591.045} C_VEL
LIN {X 0,Y 467.591,Z 245.241,A -85,B 0,C 180,E1 -7594.242,E2 -7594.242} C_VEL
LIN {X 0,Y 467.544,Z 245.245,A -85,B 0,C 180,E1 -7597.185,E2 -7597.185} C_VEL
LIN {X 0,Y 467.561,Z 245.241,A -85,B 0,C 180,E1 -7600.266,E2 -7600.266} C_VEL
LIN {X 0,Y 467.549,Z 245.245,A -85,B 0,C 180,E1 -7603.745,E2 -7603.745} C_VEL
LIN {X 0,Y 467.556,Z 245.247,A -85,B 0,C 180,E1 -7606.255,E2 -7606.255} C_VEL
LIN {X 0,Y 467.581,Z 245.243,A -85,B 0,C 180,E1 -7608.723,E2 -7608.723} C_VEL
LIN {X 0,Y 467.624,Z 245.288,A -85,B 0,C 180,E1 -7611.024,E2 -7611.024} C_VEL
LIN {X 0,Y 468.423,Z 250.416,A -85,B 0,C 180,E1 -7613.654,E2 -7613.654} C_VEL
LIN {X 0,Y 468.488,Z 254.417,A -85,B 0,C 180,E1 -7615.597,E2 -7615.597} C_VEL
